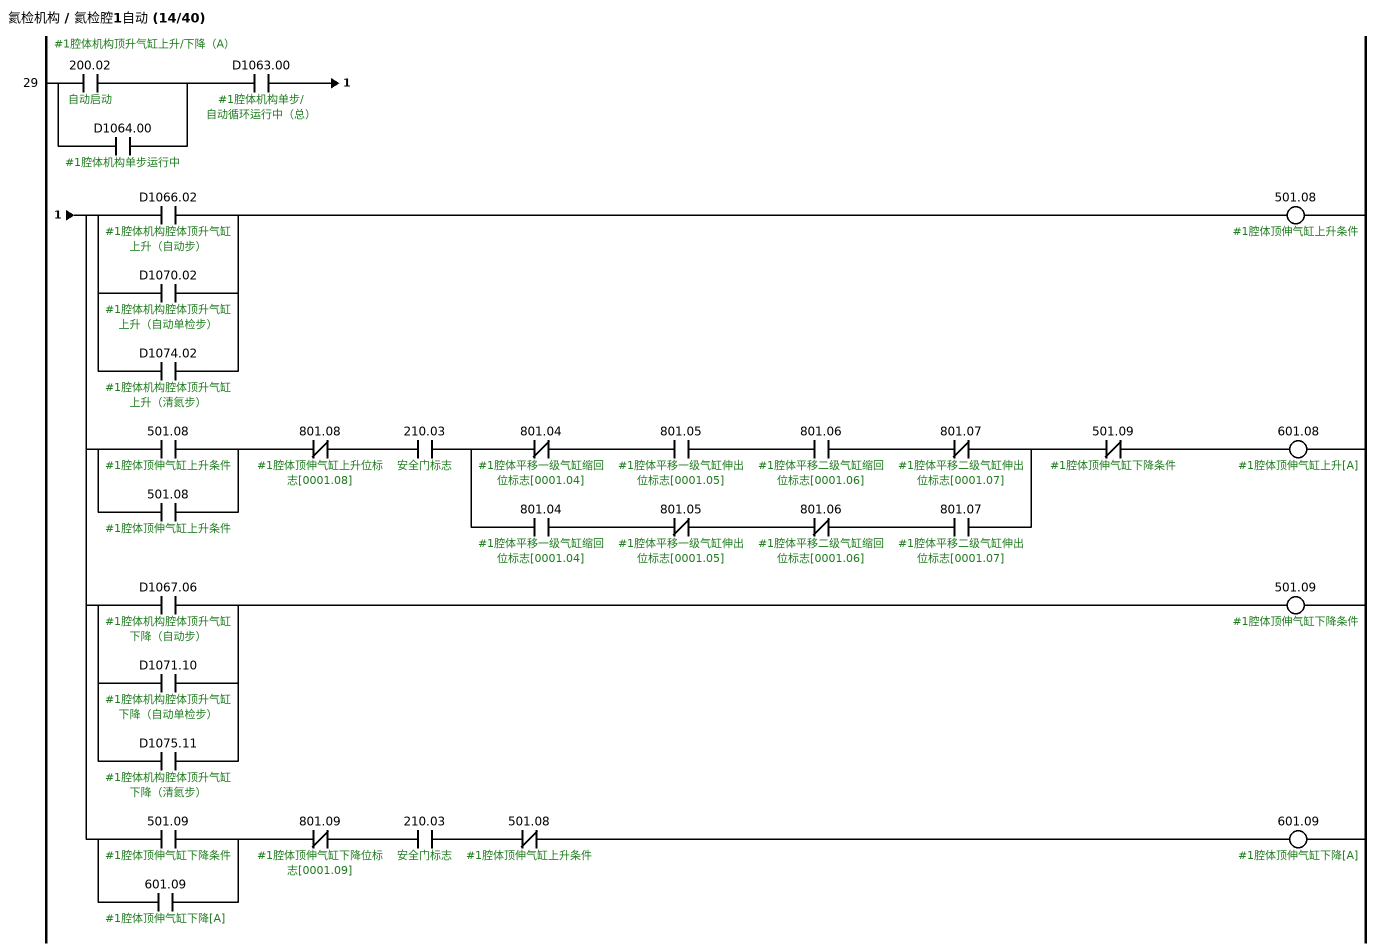
; [picture p216: 氦检机构 / 氦检腔1自动, rungs 29-29]
; rung 29: #1腔体机构顶升气缸上升/下降（A）
LD 200.02  ; 自动启动
OR D1064.00  ; #1腔体机构单步运行中
AND D1063.00  ; #1腔体机构单步/自动循环运行中（总）
OUT TR0
LD D1066.02  ; #1腔体机构腔体顶升气缸上升（自动步）
OR D1070.02  ; #1腔体机构腔体顶升气缸上升（自动单检步）
OR D1074.02  ; #1腔体机构腔体顶升气缸上升（清氦步）
ANDLD
OUT 501.08  ; #1腔体顶伸气缸上升条件
LD TR0
LD 501.08  ; #1腔体顶伸气缸上升条件
OR 501.08  ; #1腔体顶伸气缸上升条件
ANDLD
ANDNOT 801.08  ; #1腔体顶伸气缸上升位标志[0001.08]
AND 210.03  ; 安全门标志
LDNOT 801.04  ; #1腔体平移一级气缸缩回位标志[0001.04]
AND 801.05  ; #1腔体平移一级气缸伸出位标志[0001.05]
AND 801.06  ; #1腔体平移二级气缸缩回位标志[0001.06]
ANDNOT 801.07  ; #1腔体平移二级气缸伸出位标志[0001.07]
LD 801.04  ; #1腔体平移一级气缸缩回位标志[0001.04]
ANDNOT 801.05  ; #1腔体平移一级气缸伸出位标志[0001.05]
ANDNOT 801.06  ; #1腔体平移二级气缸缩回位标志[0001.06]
AND 801.07  ; #1腔体平移二级气缸伸出位标志[0001.07]
ORLD
ANDLD
ANDNOT 501.09  ; #1腔体顶伸气缸下降条件
OUT 601.08  ; #1腔体顶伸气缸上升[A]
LD TR0
LD D1067.06  ; #1腔体机构腔体顶升气缸下降（自动步）
OR D1071.10  ; #1腔体机构腔体顶升气缸下降（自动单检步）
OR D1075.11  ; #1腔体机构腔体顶升气缸下降（清氦步）
ANDLD
OUT 501.09  ; #1腔体顶伸气缸下降条件
LD TR0
LD 501.09  ; #1腔体顶伸气缸下降条件
OR 601.09  ; #1腔体顶伸气缸下降[A]
ANDLD
ANDNOT 801.09  ; #1腔体顶伸气缸下降位标志[0001.09]
AND 210.03  ; 安全门标志
ANDNOT 501.08  ; #1腔体顶伸气缸上升条件
OUT 601.09  ; #1腔体顶伸气缸下降[A]

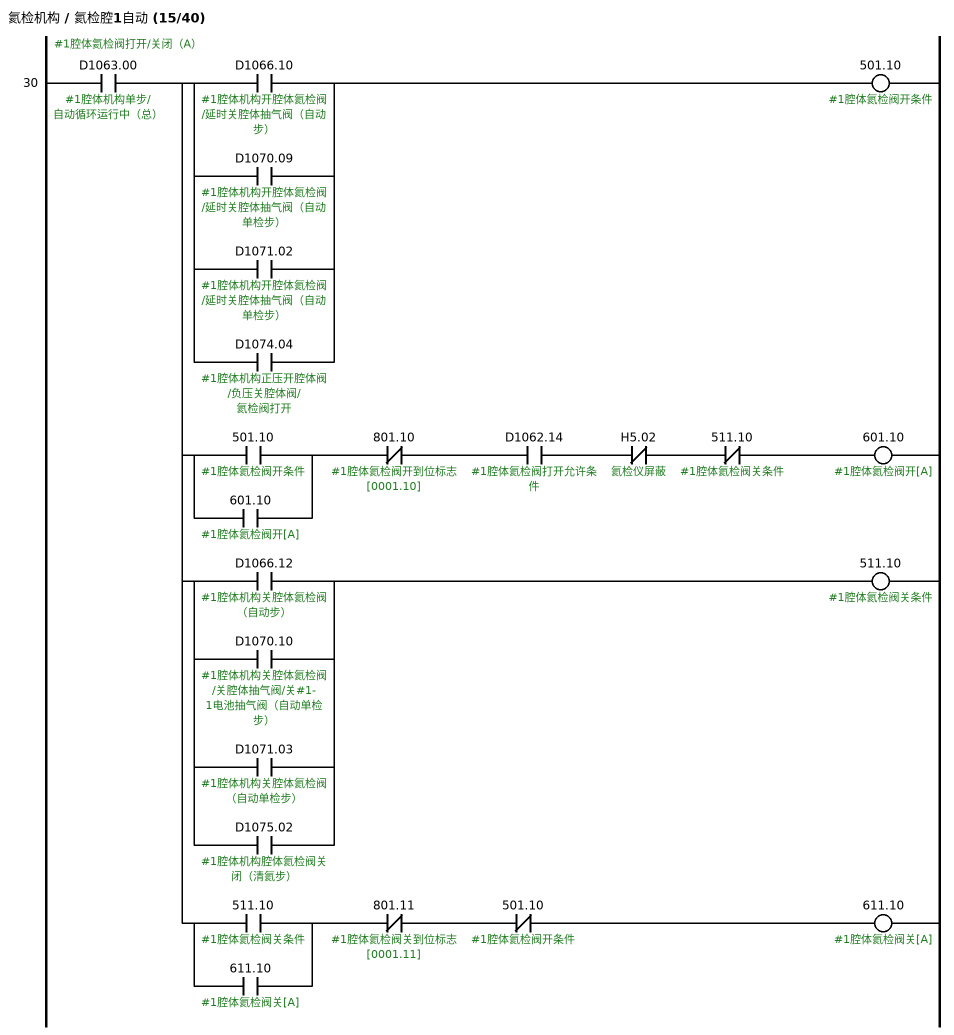
; rung 30: #1腔体氦检阀打开/关闭（A）
LD D1063.00  ; #1腔体机构单步/自动循环运行中（总）
OUT TR0
LD D1066.10  ; #1腔体机构开腔体氦检阀/延时关腔体抽气阀（自动步）
OR D1070.09  ; #1腔体机构开腔体氦检阀/延时关腔体抽气阀（自动单检步）
OR D1071.02  ; #1腔体机构开腔体氦检阀/延时关腔体抽气阀（自动单检步）
OR D1074.04  ; #1腔体机构正压开腔体阀/负压关腔体阀/氦检阀打开
ANDLD
OUT 501.10  ; #1腔体氦检阀开条件
LD TR0
LD 501.10  ; #1腔体氦检阀开条件
OR 601.10  ; #1腔体氦检阀开[A]
ANDLD
ANDNOT 801.10  ; #1腔体氦检阀开到位标志[0001.10]
AND D1062.14  ; #1腔体氦检阀打开允许条件
ANDNOT H5.02  ; 氦检仪屏蔽
ANDNOT 511.10  ; #1腔体氦检阀关条件
OUT 601.10  ; #1腔体氦检阀开[A]
LD TR0
LD D1066.12  ; #1腔体机构关腔体氦检阀（自动步）
OR D1070.10  ; #1腔体机构关腔体氦检阀/关腔体抽气阀/关#1-1电池抽气阀（自动单检步）
OR D1071.03  ; #1腔体机构关腔体氦检阀（自动单检步）
OR D1075.02  ; #1腔体机构腔体氦检阀关闭（清氦步）
ANDLD
OUT 511.10  ; #1腔体氦检阀关条件
LD TR0
LD 511.10  ; #1腔体氦检阀关条件
OR 611.10  ; #1腔体氦检阀关[A]
ANDLD
ANDNOT 801.11  ; #1腔体氦检阀关到位标志[0001.11]
ANDNOT 501.10  ; #1腔体氦检阀开条件
OUT 611.10  ; #1腔体氦检阀关[A]

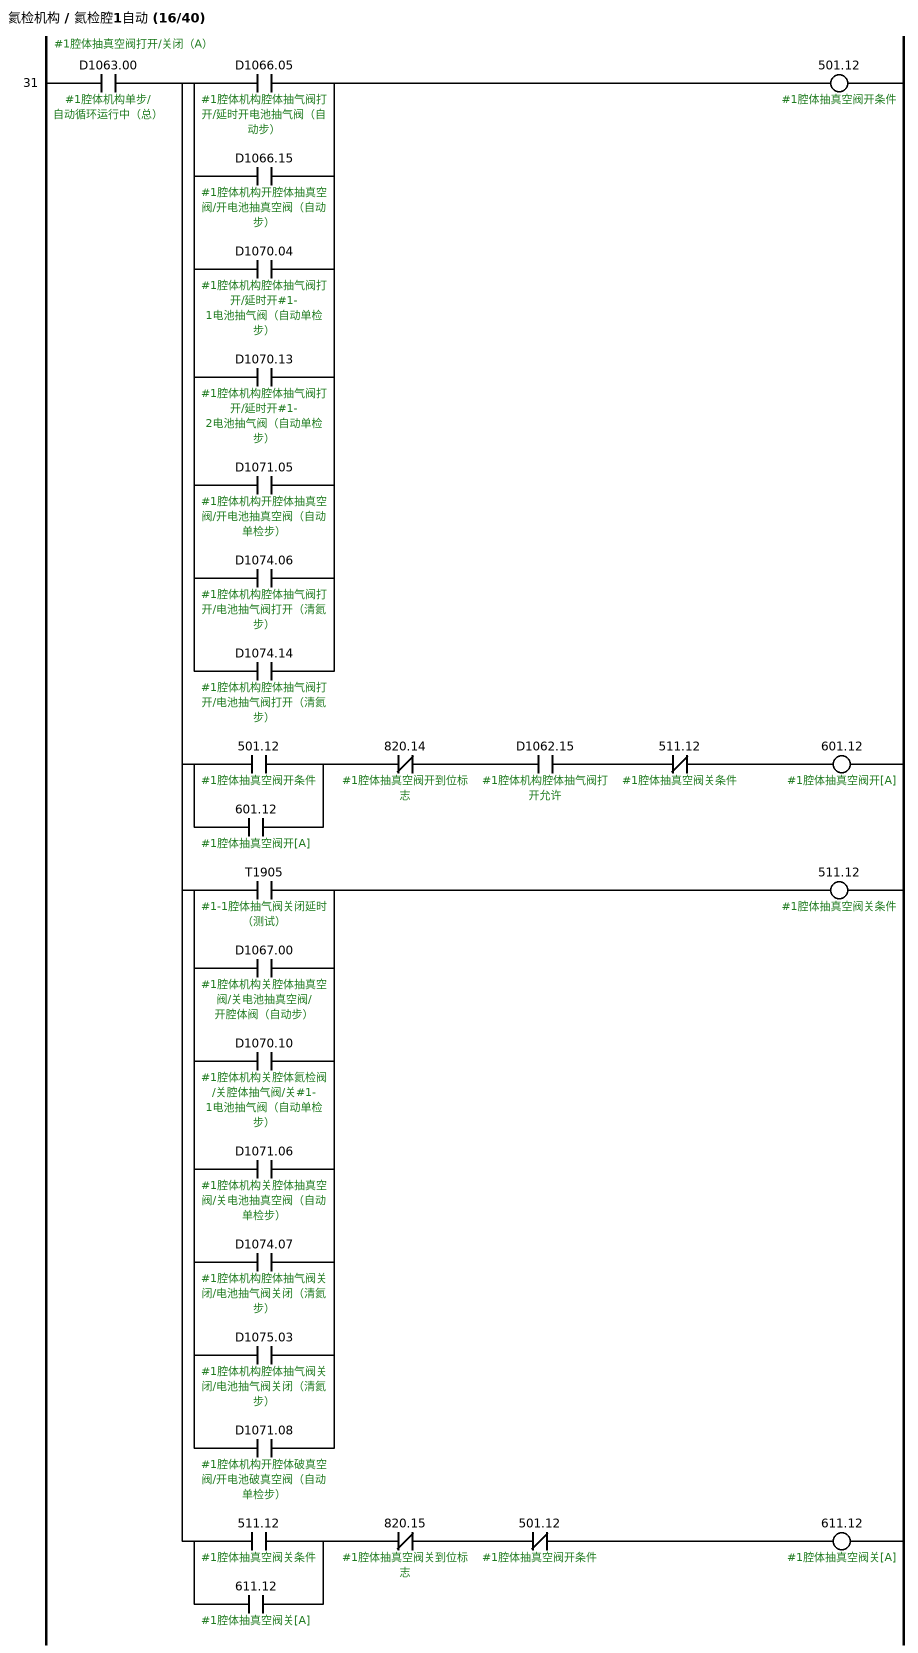
; rung 31: #1腔体抽真空阀打开/关闭（A）
LD D1063.00  ; #1腔体机构单步/自动循环运行中（总）
OUT TR0
LD D1066.05  ; #1腔体机构腔体抽气阀打开/延时开电池抽气阀（自动步）
OR D1066.15  ; #1腔体机构开腔体抽真空阀/开电池抽真空阀（自动步）
OR D1070.04  ; #1腔体机构腔体抽气阀打开/延时开#1-1电池抽气阀（自动单检步）
OR D1070.13  ; #1腔体机构腔体抽气阀打开/延时开#1-2电池抽气阀（自动单检步）
OR D1071.05  ; #1腔体机构开腔体抽真空阀/开电池抽真空阀（自动单检步）
OR D1074.06  ; #1腔体机构腔体抽气阀打开/电池抽气阀打开（清氦步）
OR D1074.14  ; #1腔体机构腔体抽气阀打开/电池抽气阀打开（清氦步）
ANDLD
OUT 501.12  ; #1腔体抽真空阀开条件
LD TR0
LD 501.12  ; #1腔体抽真空阀开条件
OR 601.12  ; #1腔体抽真空阀开[A]
ANDLD
ANDNOT 820.14  ; #1腔体抽真空阀开到位标志
AND D1062.15  ; #1腔体机构腔体抽气阀打开允许
ANDNOT 511.12  ; #1腔体抽真空阀关条件
OUT 601.12  ; #1腔体抽真空阀开[A]
LD TR0
LD T1905  ; #1-1腔体抽气阀关闭延时（测试）
OR D1067.00  ; #1腔体机构关腔体抽真空阀/关电池抽真空阀/开腔体阀（自动步）
OR D1070.10  ; #1腔体机构关腔体氦检阀/关腔体抽气阀/关#1-1电池抽气阀（自动单检步）
OR D1071.06  ; #1腔体机构关腔体抽真空阀/关电池抽真空阀（自动单检步）
OR D1074.07  ; #1腔体机构腔体抽气阀关闭/电池抽气阀关闭（清氦步）
OR D1075.03  ; #1腔体机构腔体抽气阀关闭/电池抽气阀关闭（清氦步）
OR D1071.08  ; #1腔体机构开腔体破真空阀/开电池破真空阀（自动单检步）
ANDLD
OUT 511.12  ; #1腔体抽真空阀关条件
LD TR0
LD 511.12  ; #1腔体抽真空阀关条件
OR 611.12  ; #1腔体抽真空阀关[A]
ANDLD
ANDNOT 820.15  ; #1腔体抽真空阀关到位标志
ANDNOT 501.12  ; #1腔体抽真空阀开条件
OUT 611.12  ; #1腔体抽真空阀关[A]

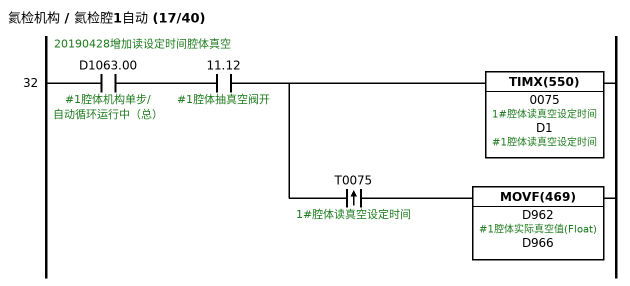
; rung 32: 20190428增加读设定时间腔体真空
LD D1063.00  ; #1腔体机构单步/自动循环运行中（总）
AND 11.12  ; #1腔体抽真空阀开
TIMX(550) 0075 D1  ; #1腔体读真空设定时间, 1#腔体读真空设定时间
@AND T0075  ; 1#腔体读真空设定时间
MOVF(469) D962 D966  ; #1腔体实际真空值(Float)

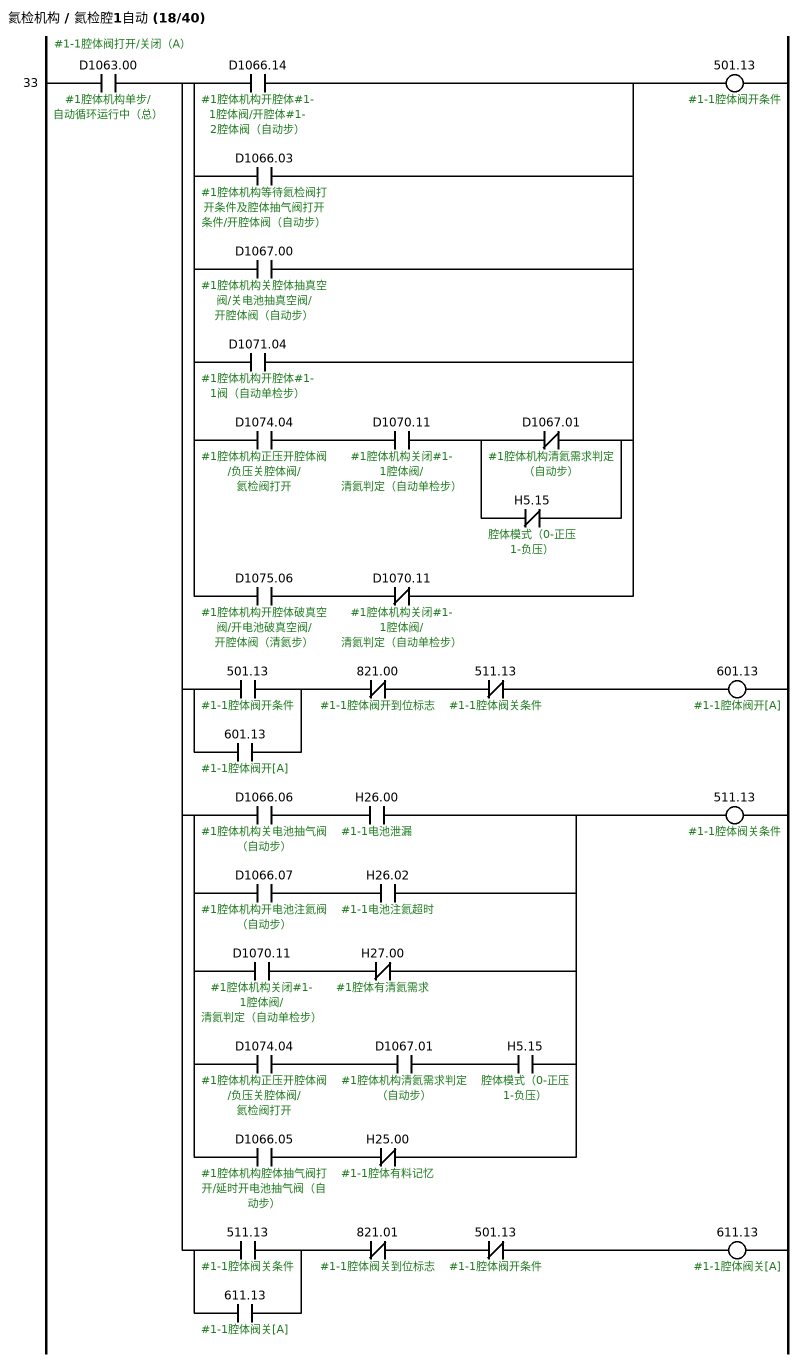
; rung 33: #1-1腔体阀打开/关闭（A）
LD D1063.00  ; #1腔体机构单步/自动循环运行中（总）
OUT TR0
LD D1066.14  ; #1腔体机构开腔体#1-1腔体阀/开腔体#1-2腔体阀（自动步）
OR D1066.03  ; #1腔体机构等待氦检阀打开条件及腔体抽气阀打开条件/开腔体阀（自动步）
OR D1067.00  ; #1腔体机构关腔体抽真空阀/关电池抽真空阀/开腔体阀（自动步）
OR D1071.04  ; #1腔体机构开腔体#1-1阀（自动单检步）
LD D1074.04  ; #1腔体机构正压开腔体阀/负压关腔体阀/氦检阀打开
AND D1070.11  ; #1腔体机构关闭#1-1腔体阀/清氦判定（自动单检步）
LDNOT D1067.01  ; #1腔体机构清氦需求判定（自动步）
ORNOT H5.15  ; 腔体模式（0-正压 1-负压）
ANDLD
ORLD
LD D1075.06  ; #1腔体机构开腔体破真空阀/开电池破真空阀/开腔体阀（清氦步）
ANDNOT D1070.11  ; #1腔体机构关闭#1-1腔体阀/清氦判定（自动单检步）
ORLD
ANDLD
OUT 501.13  ; #1-1腔体阀开条件
LD TR0
LD 501.13  ; #1-1腔体阀开条件
OR 601.13  ; #1-1腔体阀开[A]
ANDLD
ANDNOT 821.00  ; #1-1腔体阀开到位标志
ANDNOT 511.13  ; #1-1腔体阀关条件
OUT 601.13  ; #1-1腔体阀开[A]
LD TR0
LD D1066.06  ; #1腔体机构关电池抽气阀（自动步）
AND H26.00  ; #1-1电池泄漏
LD D1066.07  ; #1腔体机构开电池注氦阀（自动步）
AND H26.02  ; #1-1电池注氦超时
ORLD
LD D1070.11  ; #1腔体机构关闭#1-1腔体阀/清氦判定（自动单检步）
ANDNOT H27.00  ; #1腔体有清氦需求
ORLD
LD D1074.04  ; #1腔体机构正压开腔体阀/负压关腔体阀/氦检阀打开
AND D1067.01  ; #1腔体机构清氦需求判定（自动步）
AND H5.15  ; 腔体模式（0-正压 1-负压）
ORLD
LD D1066.05  ; #1腔体机构腔体抽气阀打开/延时开电池抽气阀（自动步）  // #1-1无料时不测试
ANDNOT H25.00  ; #1-1腔体有料记忆
ORLD
ANDLD
OUT 511.13  ; #1-1腔体阀关条件
LD TR0
LD 511.13  ; #1-1腔体阀关条件
OR 611.13  ; #1-1腔体阀关[A]
ANDLD
ANDNOT 821.01  ; #1-1腔体阀关到位标志
ANDNOT 501.13  ; #1-1腔体阀开条件
OUT 611.13  ; #1-1腔体阀关[A]

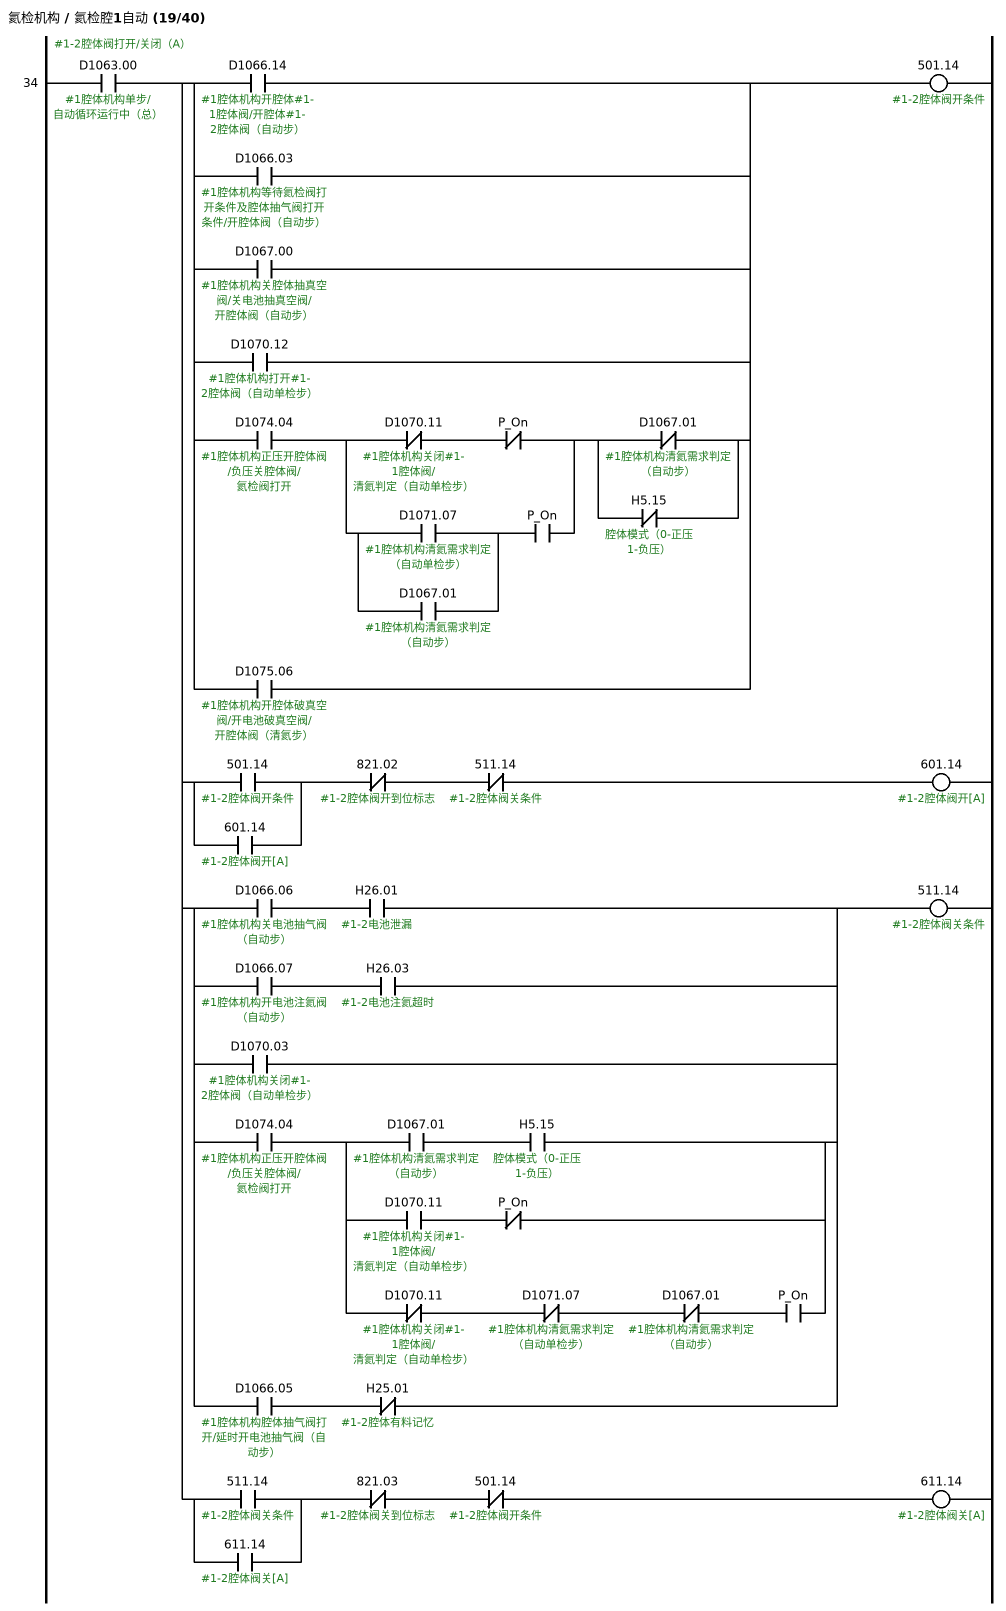
; rung 34: #1-2腔体阀打开/关闭（A）
LD D1063.00  ; #1腔体机构单步/自动循环运行中（总）
OUT TR0
LD D1066.14  ; #1腔体机构开腔体#1-1腔体阀/开腔体#1-2腔体阀（自动步）
OR D1066.03  ; #1腔体机构等待氦检阀打开条件及腔体抽气阀打开条件/开腔体阀（自动步）
OR D1067.00  ; #1腔体机构关腔体抽真空阀/关电池抽真空阀/开腔体阀（自动步）
OR D1070.12  ; #1腔体机构打开#1-2腔体阀（自动单检步）
LD D1074.04  ; #1腔体机构正压开腔体阀/负压关腔体阀/氦检阀打开
LDNOT D1070.11  ; #1腔体机构关闭#1-1腔体阀/清氦判定（自动单检步）
ANDNOT P_On
LD D1071.07  ; #1腔体机构清氦需求判定（自动单检步）
OR D1067.01  ; #1腔体机构清氦需求判定（自动步）
AND P_On
ORLD
ANDLD
LDNOT D1067.01  ; #1腔体机构清氦需求判定（自动步）
ORNOT H5.15  ; 腔体模式（0-正压 1-负压）
ANDLD
ORLD
OR D1075.06  ; #1腔体机构开腔体破真空阀/开电池破真空阀/开腔体阀（清氦步）
ANDLD
OUT 501.14  ; #1-2腔体阀开条件
LD TR0
LD 501.14  ; #1-2腔体阀开条件
OR 601.14  ; #1-2腔体阀开[A]
ANDLD
ANDNOT 821.02  ; #1-2腔体阀开到位标志
ANDNOT 511.14  ; #1-2腔体阀关条件
OUT 601.14  ; #1-2腔体阀开[A]
LD TR0
LD D1066.06  ; #1腔体机构关电池抽气阀（自动步）
AND H26.01  ; #1-2电池泄漏
LD D1066.07  ; #1腔体机构开电池注氦阀（自动步）
AND H26.03  ; #1-2电池注氦超时
ORLD
OR D1070.03  ; #1腔体机构关闭#1-2腔体阀（自动单检步）
LD D1074.04  ; #1腔体机构正压开腔体阀/负压关腔体阀/氦检阀打开
LD D1067.01  ; #1腔体机构清氦需求判定（自动步）
AND H5.15  ; 腔体模式（0-正压 1-负压）
LD D1070.11  ; #1腔体机构关闭#1-1腔体阀/清氦判定（自动单检步）
ANDNOT P_On
ORLD
LDNOT D1070.11  ; #1腔体机构关闭#1-1腔体阀/清氦判定（自动单检步）
ANDNOT D1071.07  ; #1腔体机构清氦需求判定（自动单检步）
ANDNOT D1067.01  ; #1腔体机构清氦需求判定（自动步）
AND P_On
ORLD
ANDLD
ORLD
LD D1066.05  ; #1腔体机构腔体抽气阀打开/延时开电池抽气阀（自动步）  // #1-2无料时不测试
ANDNOT H25.01  ; #1-2腔体有料记忆
ORLD
ANDLD
OUT 511.14  ; #1-2腔体阀关条件
LD TR0
LD 511.14  ; #1-2腔体阀关条件
OR 611.14  ; #1-2腔体阀关[A]
ANDLD
ANDNOT 821.03  ; #1-2腔体阀关到位标志
ANDNOT 501.14  ; #1-2腔体阀开条件
OUT 611.14  ; #1-2腔体阀关[A]

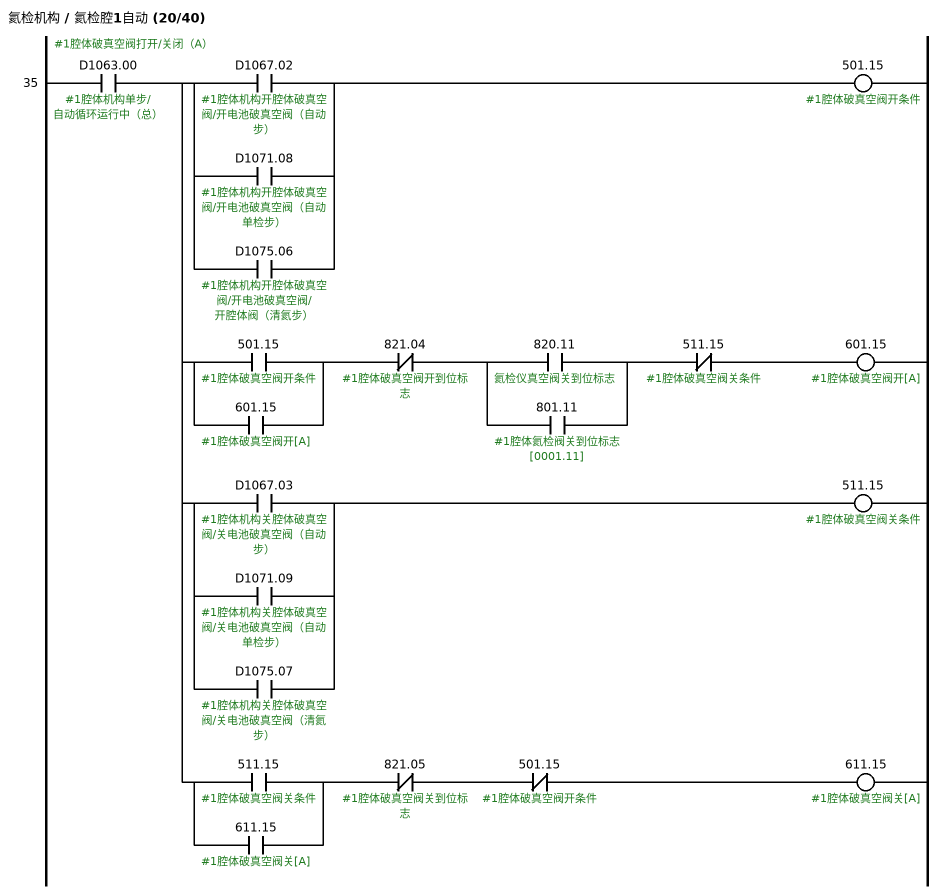
; rung 35: #1腔体破真空阀打开/关闭（A）
LD D1063.00  ; #1腔体机构单步/自动循环运行中（总）
OUT TR0
LD D1067.02  ; #1腔体机构开腔体破真空阀/开电池破真空阀（自动步）
OR D1071.08  ; #1腔体机构开腔体破真空阀/开电池破真空阀（自动单检步）
OR D1075.06  ; #1腔体机构开腔体破真空阀/开电池破真空阀/开腔体阀（清氦步）
ANDLD
OUT 501.15  ; #1腔体破真空阀开条件
LD TR0
LD 501.15  ; #1腔体破真空阀开条件
OR 601.15  ; #1腔体破真空阀开[A]
ANDLD
ANDNOT 821.04  ; #1腔体破真空阀开到位标志
LD 820.11  ; 氦检仪真空阀关到位标志
OR 801.11  ; #1腔体氦检阀关到位标志[0001.11]
ANDLD
ANDNOT 511.15  ; #1腔体破真空阀关条件
OUT 601.15  ; #1腔体破真空阀开[A]
LD TR0
LD D1067.03  ; #1腔体机构关腔体破真空阀/关电池破真空阀（自动步）
OR D1071.09  ; #1腔体机构关腔体破真空阀/关电池破真空阀（自动单检步）
OR D1075.07  ; #1腔体机构关腔体破真空阀/关电池破真空阀（清氦步）
ANDLD
OUT 511.15  ; #1腔体破真空阀关条件
LD TR0
LD 511.15  ; #1腔体破真空阀关条件
OR 611.15  ; #1腔体破真空阀关[A]
ANDLD
ANDNOT 821.05  ; #1腔体破真空阀关到位标志
ANDNOT 501.15  ; #1腔体破真空阀开条件
OUT 611.15  ; #1腔体破真空阀关[A]

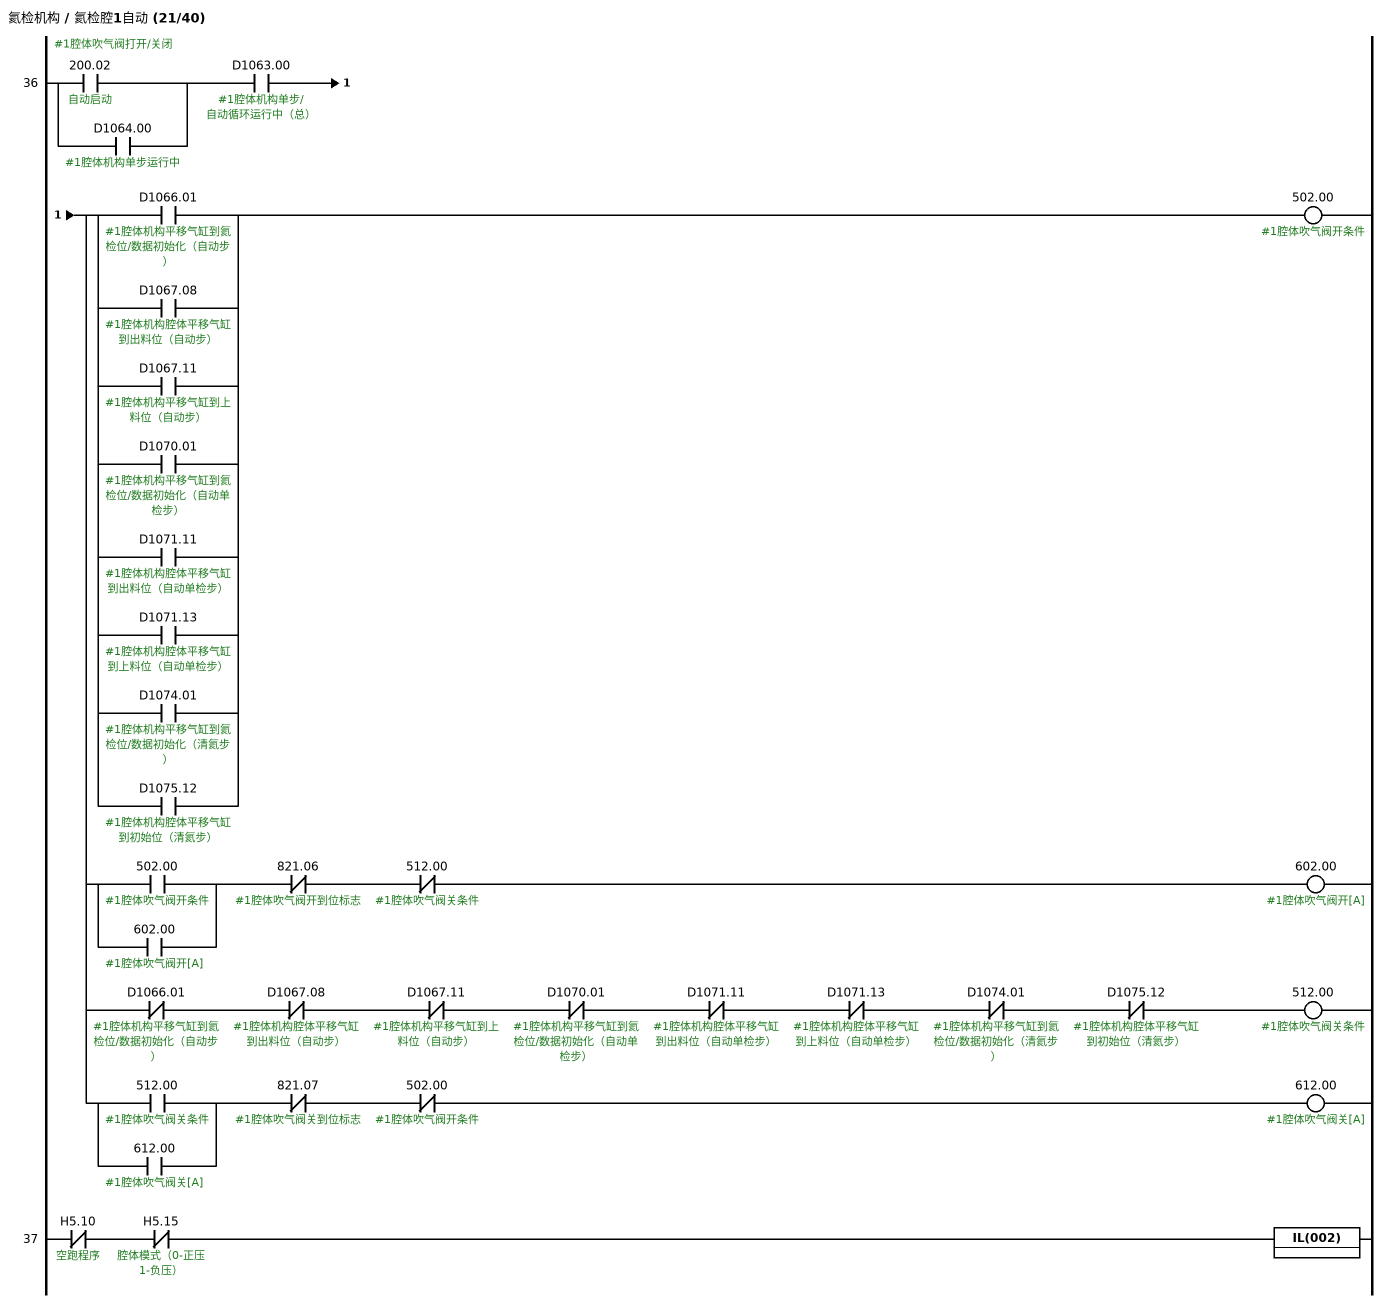
; rung 36: #1腔体吹气阀打开/关闭
LD 200.02  ; 自动启动
OR D1064.00  ; #1腔体机构单步运行中
AND D1063.00  ; #1腔体机构单步/自动循环运行中（总）
OUT TR0
LD D1066.01  ; #1腔体机构平移气缸到氦检位/数据初始化（自动步）
OR D1067.08  ; #1腔体机构腔体平移气缸到出料位（自动步）
OR D1067.11  ; #1腔体机构平移气缸到上料位（自动步）
OR D1070.01  ; #1腔体机构平移气缸到氦检位/数据初始化（自动单检步）
OR D1071.11  ; #1腔体机构腔体平移气缸到出料位（自动单检步）
OR D1071.13  ; #1腔体机构腔体平移气缸到上料位（自动单检步）
OR D1074.01  ; #1腔体机构平移气缸到氦检位/数据初始化（清氦步）
OR D1075.12  ; #1腔体机构腔体平移气缸到初始位（清氦步）
ANDLD
OUT 502.00  ; #1腔体吹气阀开条件
LD TR0
LD 502.00  ; #1腔体吹气阀开条件
OR 602.00  ; #1腔体吹气阀开[A]
ANDLD
ANDNOT 821.06  ; #1腔体吹气阀开到位标志
ANDNOT 512.00  ; #1腔体吹气阀关条件
OUT 602.00  ; #1腔体吹气阀开[A]
LD TR0
ANDNOT D1066.01  ; #1腔体机构平移气缸到氦检位/数据初始化（自动步）
ANDNOT D1067.08  ; #1腔体机构腔体平移气缸到出料位（自动步）
ANDNOT D1067.11  ; #1腔体机构平移气缸到上料位（自动步）
ANDNOT D1070.01  ; #1腔体机构平移气缸到氦检位/数据初始化（自动单检步）
ANDNOT D1071.11  ; #1腔体机构腔体平移气缸到出料位（自动单检步）
ANDNOT D1071.13  ; #1腔体机构腔体平移气缸到上料位（自动单检步）
ANDNOT D1074.01  ; #1腔体机构平移气缸到氦检位/数据初始化（清氦步）
ANDNOT D1075.12  ; #1腔体机构腔体平移气缸到初始位（清氦步）
OUT 512.00  ; #1腔体吹气阀关条件
LD TR0
LD 512.00  ; #1腔体吹气阀关条件
OR 612.00  ; #1腔体吹气阀关[A]
ANDLD
ANDNOT 821.07  ; #1腔体吹气阀关到位标志
ANDNOT 502.00  ; #1腔体吹气阀开条件
OUT 612.00  ; #1腔体吹气阀关[A]
; rung 37
LDNOT H5.10  ; 空跑程序
ANDNOT H5.15  ; 腔体模式（0-正压 1-负压）
IL(002)

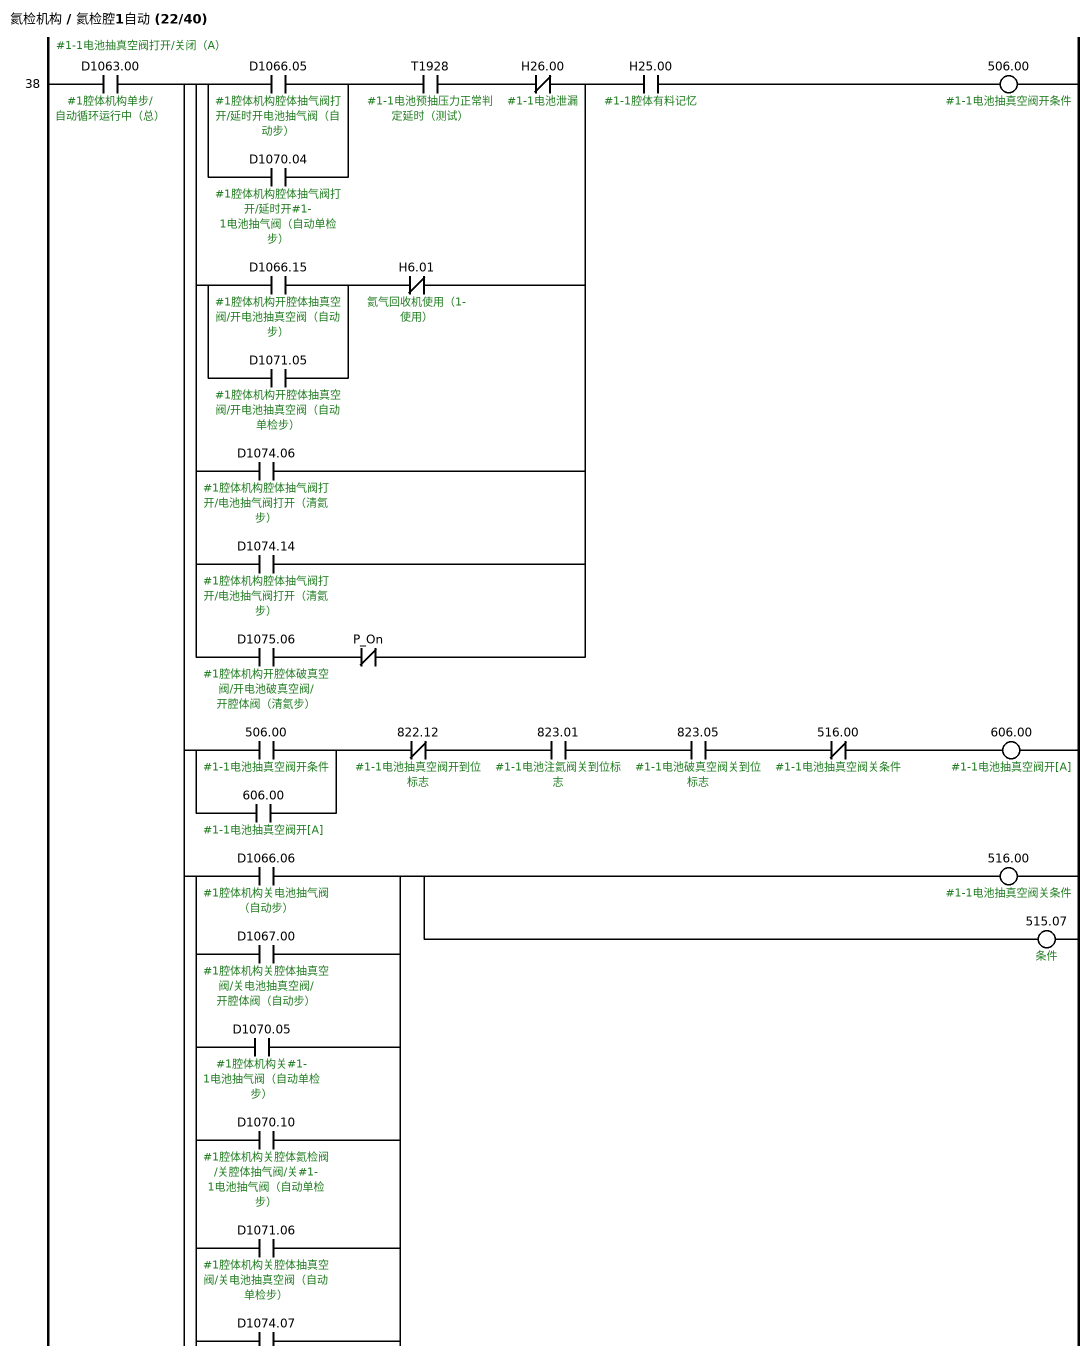

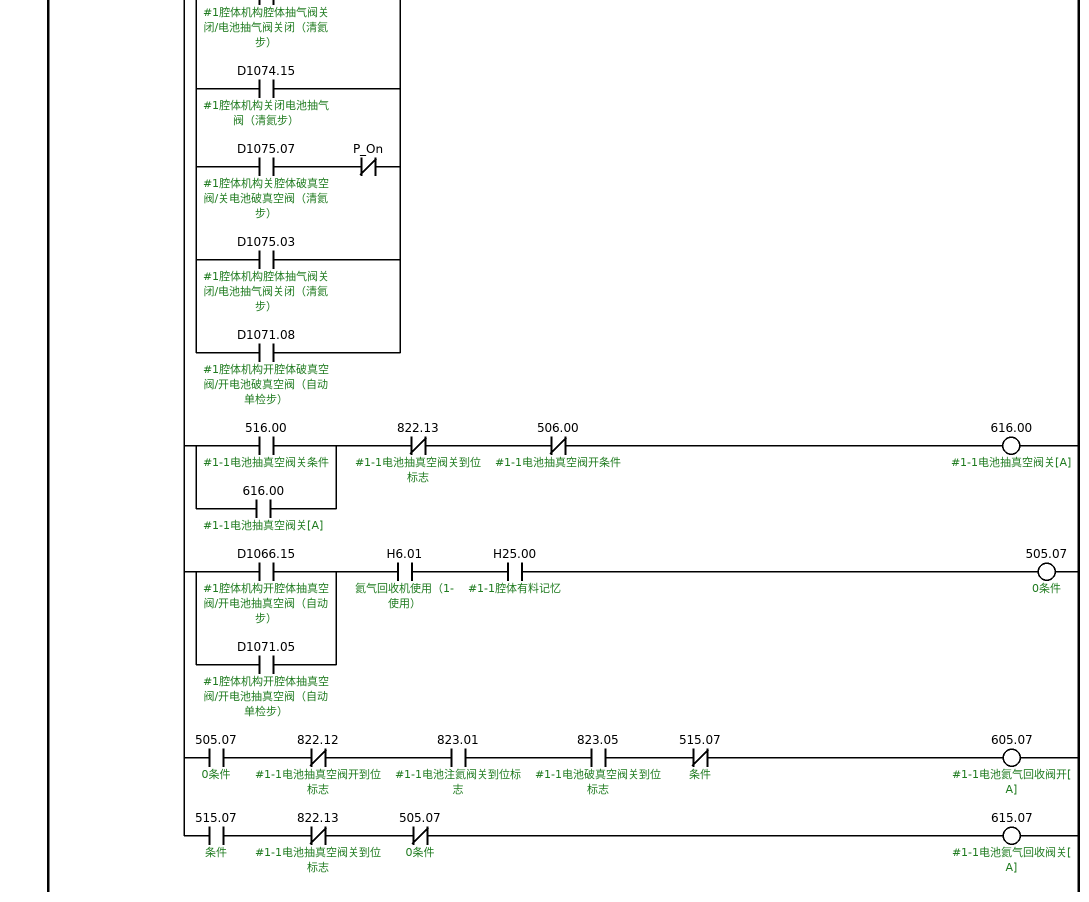
; rung 38: #1-1电池抽真空阀打开/关闭（A）
LD D1063.00  ; #1腔体机构单步/自动循环运行中（总）
OUT TR0
LD D1066.05  ; #1腔体机构腔体抽气阀打开/延时开电池抽气阀（自动步）
OR D1070.04  ; #1腔体机构腔体抽气阀打开/延时开#1-1电池抽气阀（自动单检步）
AND T1928  ; #1-1电池预抽压力正常判定延时（测试）
ANDNOT H26.00  ; #1-1电池泄漏
LD D1066.15  ; #1腔体机构开腔体抽真空阀/开电池抽真空阀（自动步）
OR D1071.05  ; #1腔体机构开腔体抽真空阀/开电池抽真空阀（自动单检步）
ANDNOT H6.01  ; 氦气回收机使用（1-使用）
ORLD
OR D1074.06  ; #1腔体机构腔体抽气阀打开/电池抽气阀打开（清氦步）
OR D1074.14  ; #1腔体机构腔体抽气阀打开/电池抽气阀打开（清氦步）
LD D1075.06  ; #1腔体机构开腔体破真空阀/开电池破真空阀/开腔体阀（清氦步）
ANDNOT P_On
ORLD
ANDLD
AND H25.00  ; #1-1腔体有料记忆
OUT 506.00  ; #1-1电池抽真空阀开条件
LD TR0
LD 506.00  ; #1-1电池抽真空阀开条件
OR 606.00  ; #1-1电池抽真空阀开[A]
ANDLD
ANDNOT 822.12  ; #1-1电池抽真空阀开到位标志
AND 823.01  ; #1-1电池注氦阀关到位标志
AND 823.05  ; #1-1电池破真空阀关到位标志
ANDNOT 516.00  ; #1-1电池抽真空阀关条件
OUT 606.00  ; #1-1电池抽真空阀开[A]
LD TR0
LD D1066.06  ; #1腔体机构关电池抽气阀（自动步）
OR D1067.00  ; #1腔体机构关腔体抽真空阀/关电池抽真空阀/开腔体阀（自动步）
OR D1070.05  ; #1腔体机构关#1-1电池抽气阀（自动单检步）
OR D1070.10  ; #1腔体机构关腔体氦检阀/关腔体抽气阀/关#1-1电池抽气阀（自动单检步）
OR D1071.06  ; #1腔体机构关腔体抽真空阀/关电池抽真空阀（自动单检步）
OR D1074.07  ; #1腔体机构腔体抽气阀关闭/电池抽气阀关闭（清氦步）
OR D1074.15  ; #1腔体机构关闭电池抽气阀（清氦步）
LD D1075.07  ; #1腔体机构关腔体破真空阀/关电池破真空阀（清氦步）
ANDNOT P_On
ORLD
OR D1075.03  ; #1腔体机构腔体抽气阀关闭/电池抽气阀关闭（清氦步）
OR D1071.08  ; #1腔体机构开腔体破真空阀/开电池破真空阀（自动单检步）
ANDLD
OUT 516.00  ; #1-1电池抽真空阀关条件
OUT 515.07  ; 条件
LD TR0
LD 516.00  ; #1-1电池抽真空阀关条件
OR 616.00  ; #1-1电池抽真空阀关[A]
ANDLD
ANDNOT 822.13  ; #1-1电池抽真空阀关到位标志
ANDNOT 506.00  ; #1-1电池抽真空阀开条件
OUT 616.00  ; #1-1电池抽真空阀关[A]
LD TR0
LD D1066.15  ; #1腔体机构开腔体抽真空阀/开电池抽真空阀（自动步）
OR D1071.05  ; #1腔体机构开腔体抽真空阀/开电池抽真空阀（自动单检步）
ANDLD
AND H6.01  ; 氦气回收机使用（1-使用）
AND H25.00  ; #1-1腔体有料记忆
OUT 505.07  ; 0条件
LD TR0
AND 505.07  ; 0条件
ANDNOT 822.12  ; #1-1电池抽真空阀开到位标志
AND 823.01  ; #1-1电池注氦阀关到位标志
AND 823.05  ; #1-1电池破真空阀关到位标志
ANDNOT 515.07  ; 条件
OUT 605.07  ; #1-1电池氦气回收阀开[A]
LD TR0
AND 515.07  ; 条件
ANDNOT 822.13  ; #1-1电池抽真空阀关到位标志
ANDNOT 505.07  ; 0条件
OUT 615.07  ; #1-1电池氦气回收阀关[A]

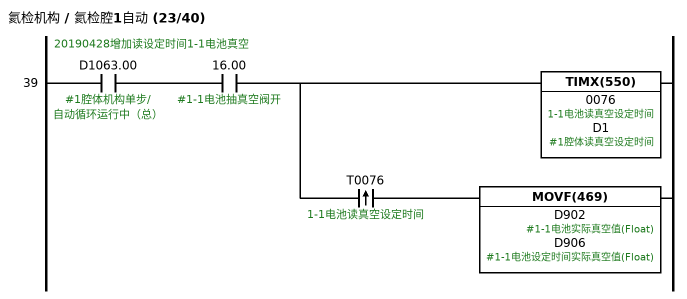
; rung 39: 20190428增加读设定时间1-1电池真空
LD D1063.00  ; #1腔体机构单步/自动循环运行中（总）
AND 16.00  ; #1-1电池抽真空阀开
TIMX(550) 0076 D1  ; #1腔体读真空设定时间, 1-1电池读真空设定时间
@AND T0076  ; 1-1电池读真空设定时间
MOVF(469) D902 D906  ; #1-1电池实际真空值(Float), #1-1电池设定时间实际真空值(Float)

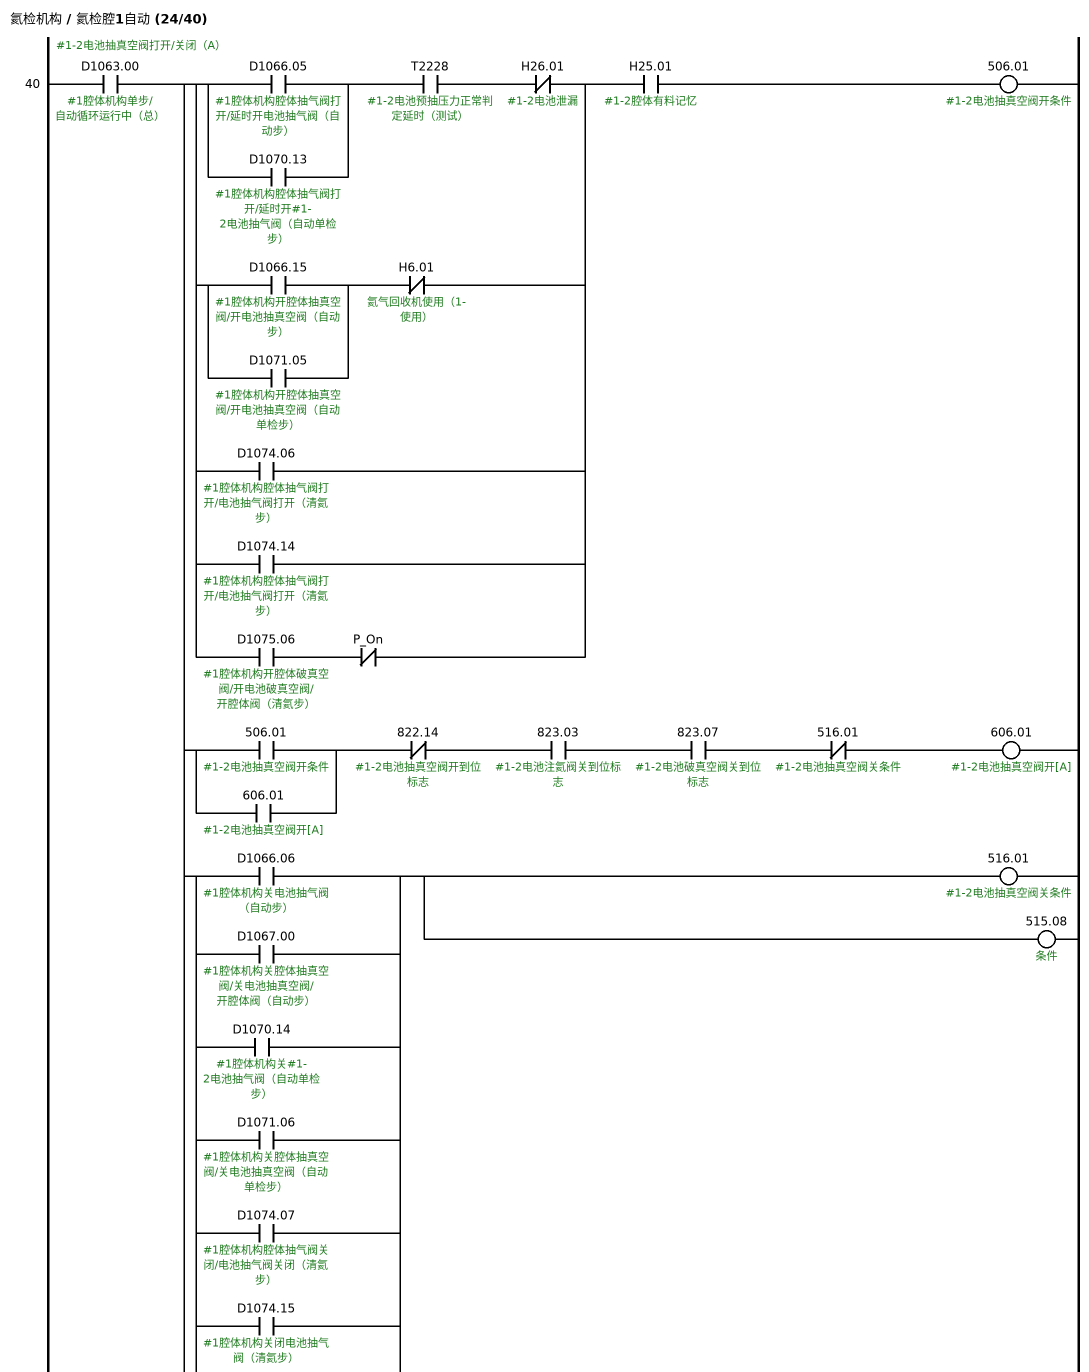

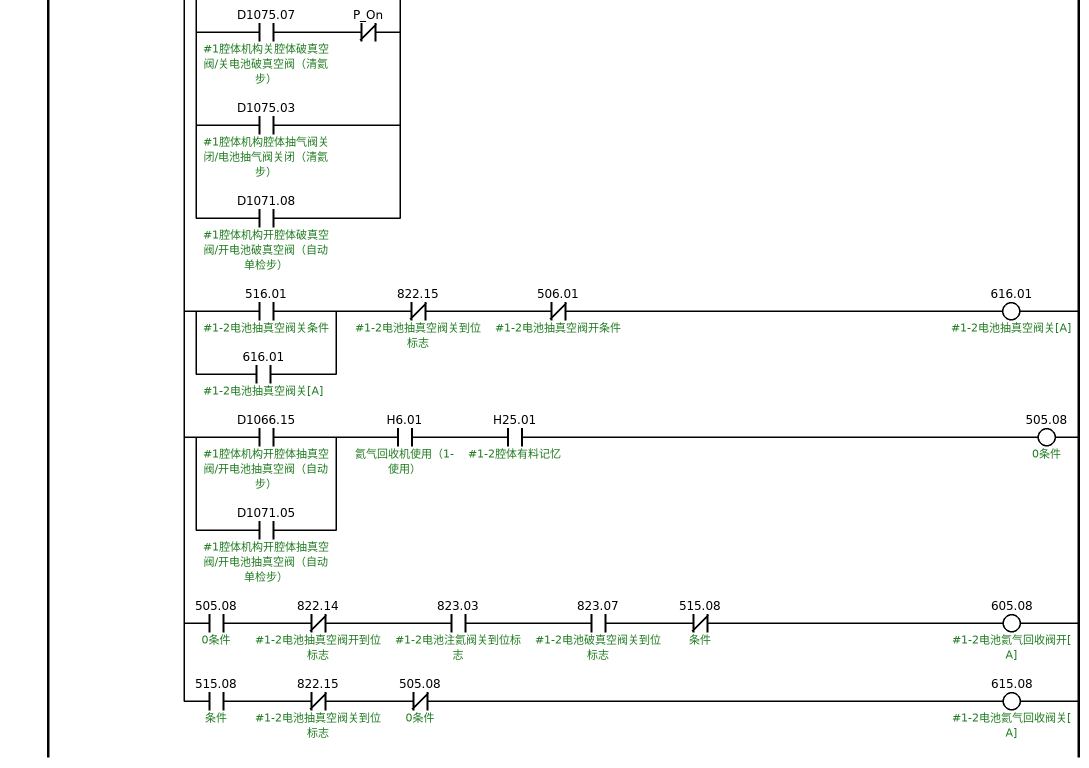
; rung 40: #1-2电池抽真空阀打开/关闭（A）
LD D1063.00  ; #1腔体机构单步/自动循环运行中（总）
OUT TR0
LD D1066.05  ; #1腔体机构腔体抽气阀打开/延时开电池抽气阀（自动步）
OR D1070.13  ; #1腔体机构腔体抽气阀打开/延时开#1-2电池抽气阀（自动单检步）
AND T2228  ; #1-2电池预抽压力正常判定延时（测试）
ANDNOT H26.01  ; #1-2电池泄漏
LD D1066.15  ; #1腔体机构开腔体抽真空阀/开电池抽真空阀（自动步）
OR D1071.05  ; #1腔体机构开腔体抽真空阀/开电池抽真空阀（自动单检步）
ANDNOT H6.01  ; 氦气回收机使用（1-使用）
ORLD
OR D1074.06  ; #1腔体机构腔体抽气阀打开/电池抽气阀打开（清氦步）
OR D1074.14  ; #1腔体机构腔体抽气阀打开/电池抽气阀打开（清氦步）
LD D1075.06  ; #1腔体机构开腔体破真空阀/开电池破真空阀/开腔体阀（清氦步）
ANDNOT P_On
ORLD
ANDLD
AND H25.01  ; #1-2腔体有料记忆
OUT 506.01  ; #1-2电池抽真空阀开条件
LD TR0
LD 506.01  ; #1-2电池抽真空阀开条件
OR 606.01  ; #1-2电池抽真空阀开[A]
ANDLD
ANDNOT 822.14  ; #1-2电池抽真空阀开到位标志
AND 823.03  ; #1-2电池注氦阀关到位标志
AND 823.07  ; #1-2电池破真空阀关到位标志
ANDNOT 516.01  ; #1-2电池抽真空阀关条件
OUT 606.01  ; #1-2电池抽真空阀开[A]
LD TR0
LD D1066.06  ; #1腔体机构关电池抽气阀（自动步）
OR D1067.00  ; #1腔体机构关腔体抽真空阀/关电池抽真空阀/开腔体阀（自动步）
OR D1070.14  ; #1腔体机构关#1-2电池抽气阀（自动单检步）
OR D1071.06  ; #1腔体机构关腔体抽真空阀/关电池抽真空阀（自动单检步）
OR D1074.07  ; #1腔体机构腔体抽气阀关闭/电池抽气阀关闭（清氦步）
OR D1074.15  ; #1腔体机构关闭电池抽气阀（清氦步）
LD D1075.07  ; #1腔体机构关腔体破真空阀/关电池破真空阀（清氦步）
ANDNOT P_On
ORLD
OR D1075.03  ; #1腔体机构腔体抽气阀关闭/电池抽气阀关闭（清氦步）
OR D1071.08  ; #1腔体机构开腔体破真空阀/开电池破真空阀（自动单检步）
ANDLD
OUT 516.01  ; #1-2电池抽真空阀关条件
OUT 515.08  ; 条件
LD TR0
LD 516.01  ; #1-2电池抽真空阀关条件
OR 616.01  ; #1-2电池抽真空阀关[A]
ANDLD
ANDNOT 822.15  ; #1-2电池抽真空阀关到位标志
ANDNOT 506.01  ; #1-2电池抽真空阀开条件
OUT 616.01  ; #1-2电池抽真空阀关[A]
LD TR0
LD D1066.15  ; #1腔体机构开腔体抽真空阀/开电池抽真空阀（自动步）
OR D1071.05  ; #1腔体机构开腔体抽真空阀/开电池抽真空阀（自动单检步）
ANDLD
AND H6.01  ; 氦气回收机使用（1-使用）
AND H25.01  ; #1-2腔体有料记忆
OUT 505.08  ; 0条件
LD TR0
AND 505.08  ; 0条件
ANDNOT 822.14  ; #1-2电池抽真空阀开到位标志
AND 823.03  ; #1-2电池注氦阀关到位标志
AND 823.07  ; #1-2电池破真空阀关到位标志
ANDNOT 515.08  ; 条件
OUT 605.08  ; #1-2电池氦气回收阀开[A]
LD TR0
AND 515.08  ; 条件
ANDNOT 822.15  ; #1-2电池抽真空阀关到位标志
ANDNOT 505.08  ; 0条件
OUT 615.08  ; #1-2电池氦气回收阀关[A]

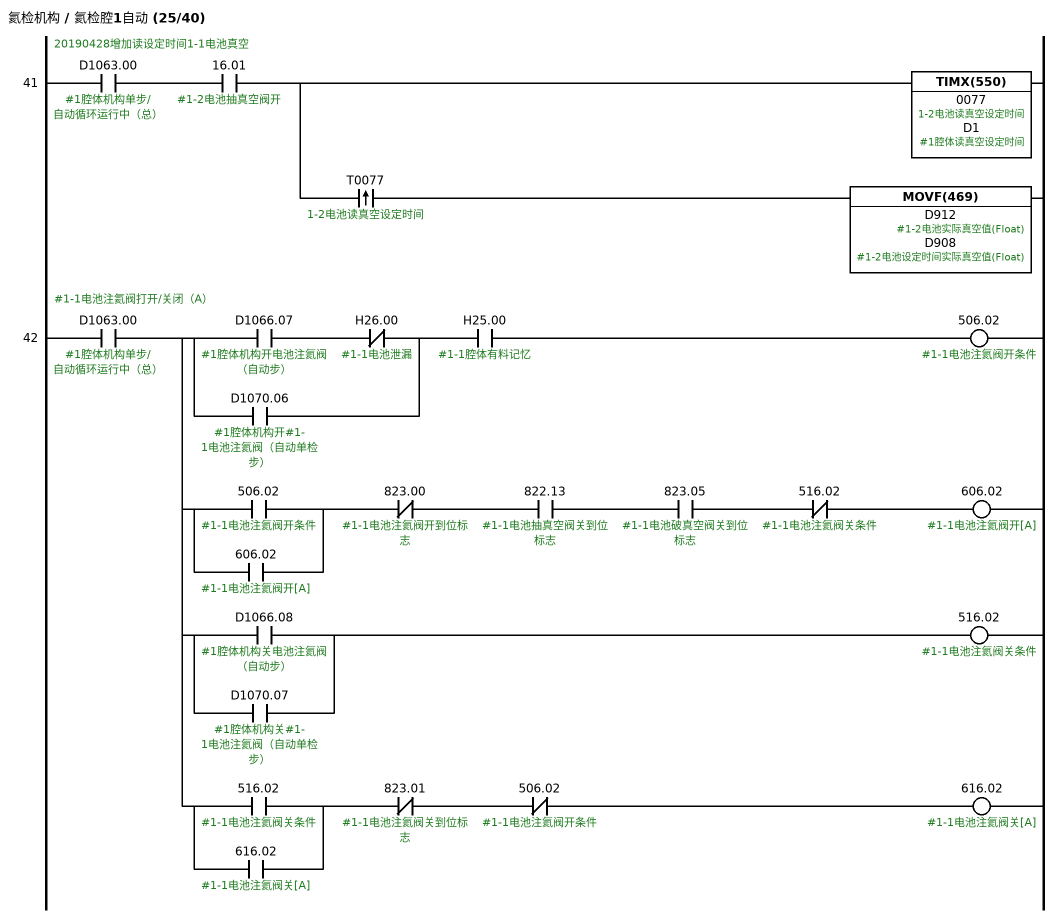
; rung 41: 20190428增加读设定时间1-1电池真空
LD D1063.00  ; #1腔体机构单步/自动循环运行中（总）
AND 16.01  ; #1-2电池抽真空阀开
TIMX(550) 0077 D1  ; #1腔体读真空设定时间, 1-2电池读真空设定时间
@AND T0077  ; 1-2电池读真空设定时间
MOVF(469) D912 D908  ; #1-2电池实际真空值(Float), #1-2电池设定时间实际真空值(Float)
; rung 42: #1-1电池注氦阀打开/关闭（A）
LD D1063.00  ; #1腔体机构单步/自动循环运行中（总）
OUT TR0
LD D1066.07  ; #1腔体机构开电池注氦阀（自动步）
ANDNOT H26.00  ; #1-1电池泄漏
OR D1070.06  ; #1腔体机构开#1-1电池注氦阀（自动单检步）
ANDLD
AND H25.00  ; #1-1腔体有料记忆
OUT 506.02  ; #1-1电池注氦阀开条件
LD TR0
LD 506.02  ; #1-1电池注氦阀开条件
OR 606.02  ; #1-1电池注氦阀开[A]
ANDLD
ANDNOT 823.00  ; #1-1电池注氦阀开到位标志
AND 822.13  ; #1-1电池抽真空阀关到位标志
AND 823.05  ; #1-1电池破真空阀关到位标志
ANDNOT 516.02  ; #1-1电池注氦阀关条件
OUT 606.02  ; #1-1电池注氦阀开[A]
LD TR0
LD D1066.08  ; #1腔体机构关电池注氦阀（自动步）
OR D1070.07  ; #1腔体机构关#1-1电池注氦阀（自动单检步）
ANDLD
OUT 516.02  ; #1-1电池注氦阀关条件
LD TR0
LD 516.02  ; #1-1电池注氦阀关条件
OR 616.02  ; #1-1电池注氦阀关[A]
ANDLD
ANDNOT 823.01  ; #1-1电池注氦阀关到位标志
ANDNOT 506.02  ; #1-1电池注氦阀开条件
OUT 616.02  ; #1-1电池注氦阀关[A]

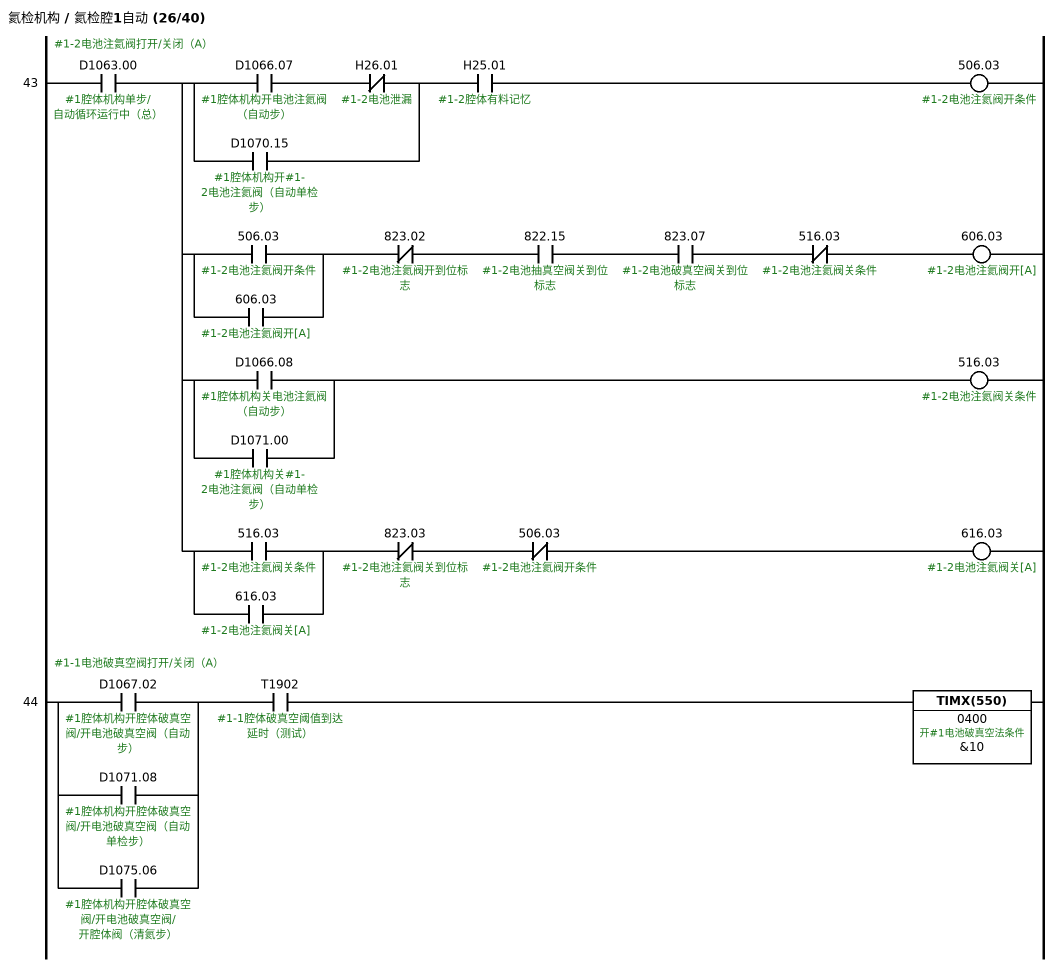
; rung 43: #1-2电池注氦阀打开/关闭（A）
LD D1063.00  ; #1腔体机构单步/自动循环运行中（总）
OUT TR0
LD D1066.07  ; #1腔体机构开电池注氦阀（自动步）
ANDNOT H26.01  ; #1-2电池泄漏
OR D1070.15  ; #1腔体机构开#1-2电池注氦阀（自动单检步）
ANDLD
AND H25.01  ; #1-2腔体有料记忆
OUT 506.03  ; #1-2电池注氦阀开条件
LD TR0
LD 506.03  ; #1-2电池注氦阀开条件
OR 606.03  ; #1-2电池注氦阀开[A]
ANDLD
ANDNOT 823.02  ; #1-2电池注氦阀开到位标志
AND 822.15  ; #1-2电池抽真空阀关到位标志
AND 823.07  ; #1-2电池破真空阀关到位标志
ANDNOT 516.03  ; #1-2电池注氦阀关条件
OUT 606.03  ; #1-2电池注氦阀开[A]
LD TR0
LD D1066.08  ; #1腔体机构关电池注氦阀（自动步）
OR D1071.00  ; #1腔体机构关#1-2电池注氦阀（自动单检步）
ANDLD
OUT 516.03  ; #1-2电池注氦阀关条件
LD TR0
LD 516.03  ; #1-2电池注氦阀关条件
OR 616.03  ; #1-2电池注氦阀关[A]
ANDLD
ANDNOT 823.03  ; #1-2电池注氦阀关到位标志
ANDNOT 506.03  ; #1-2电池注氦阀开条件
OUT 616.03  ; #1-2电池注氦阀关[A]
; rung 44: #1-1电池破真空阀打开/关闭（A）
LD D1067.02  ; #1腔体机构开腔体破真空阀/开电池破真空阀（自动步）
OR D1071.08  ; #1腔体机构开腔体破真空阀/开电池破真空阀（自动单检步）
OR D1075.06  ; #1腔体机构开腔体破真空阀/开电池破真空阀/开腔体阀（清氦步）
AND T1902  ; #1-1腔体破真空阈值到达延时（测试）
TIMX(550) 0400 &10  ; 开#1电池破真空法条件

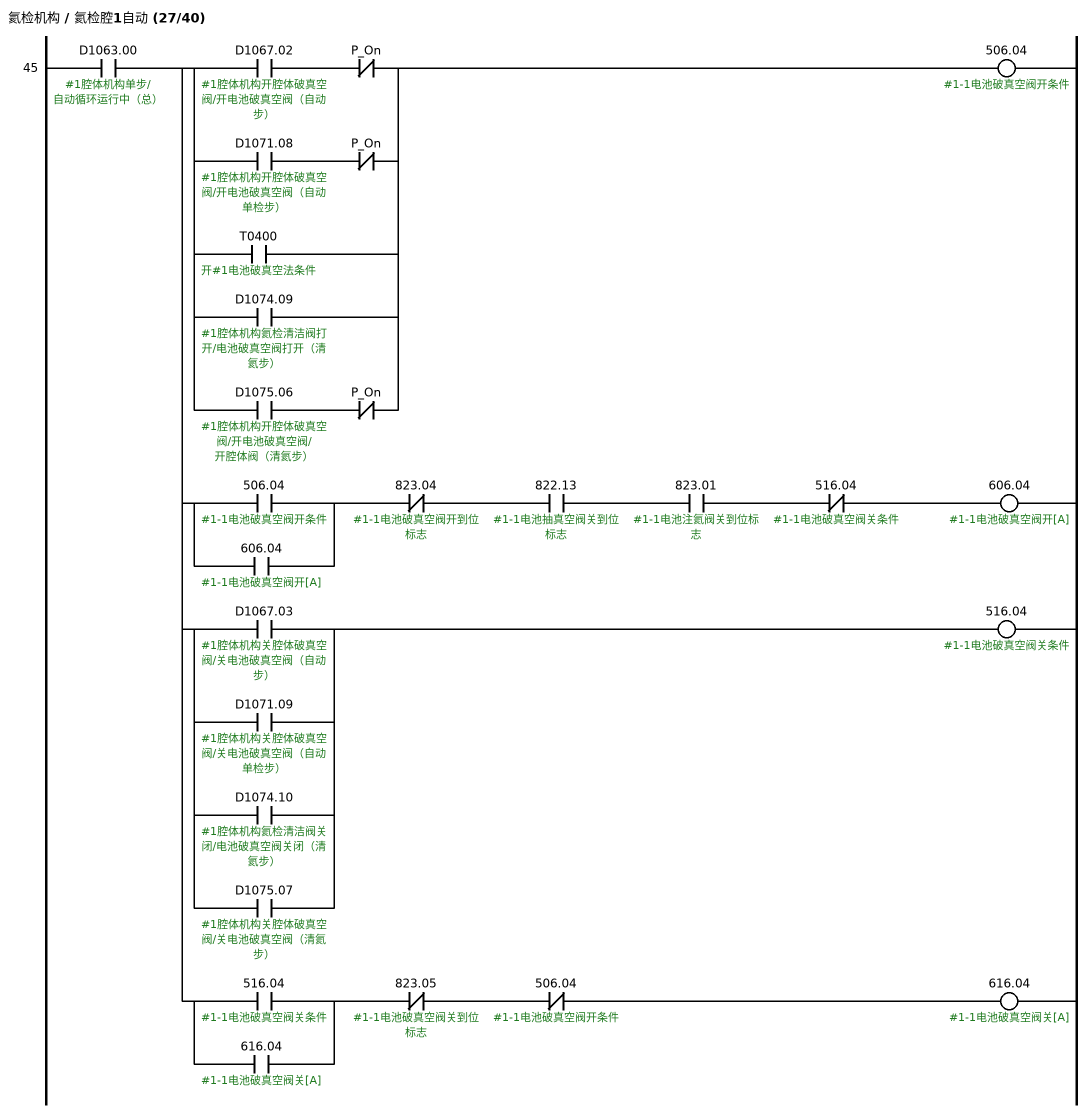
; rung 45
LD D1063.00  ; #1腔体机构单步/自动循环运行中（总）
OUT TR0
LD D1067.02  ; #1腔体机构开腔体破真空阀/开电池破真空阀（自动步）
ANDNOT P_On
LD D1071.08  ; #1腔体机构开腔体破真空阀/开电池破真空阀（自动单检步）
ANDNOT P_On
ORLD
OR T0400  ; 开#1电池破真空法条件
OR D1074.09  ; #1腔体机构氦检清洁阀打开/电池破真空阀打开（清氦步）
LD D1075.06  ; #1腔体机构开腔体破真空阀/开电池破真空阀/开腔体阀（清氦步）
ANDNOT P_On
ORLD
ANDLD
OUT 506.04  ; #1-1电池破真空阀开条件
LD TR0
LD 506.04  ; #1-1电池破真空阀开条件
OR 606.04  ; #1-1电池破真空阀开[A]
ANDLD
ANDNOT 823.04  ; #1-1电池破真空阀开到位标志
AND 822.13  ; #1-1电池抽真空阀关到位标志
AND 823.01  ; #1-1电池注氦阀关到位标志
ANDNOT 516.04  ; #1-1电池破真空阀关条件
OUT 606.04  ; #1-1电池破真空阀开[A]
LD TR0
LD D1067.03  ; #1腔体机构关腔体破真空阀/关电池破真空阀（自动步）
OR D1071.09  ; #1腔体机构关腔体破真空阀/关电池破真空阀（自动单检步）
OR D1074.10  ; #1腔体机构氦检清洁阀关闭/电池破真空阀关闭（清氦步）
OR D1075.07  ; #1腔体机构关腔体破真空阀/关电池破真空阀（清氦步）
ANDLD
OUT 516.04  ; #1-1电池破真空阀关条件
LD TR0
LD 516.04  ; #1-1电池破真空阀关条件
OR 616.04  ; #1-1电池破真空阀关[A]
ANDLD
ANDNOT 823.05  ; #1-1电池破真空阀关到位标志
ANDNOT 506.04  ; #1-1电池破真空阀开条件
OUT 616.04  ; #1-1电池破真空阀关[A]

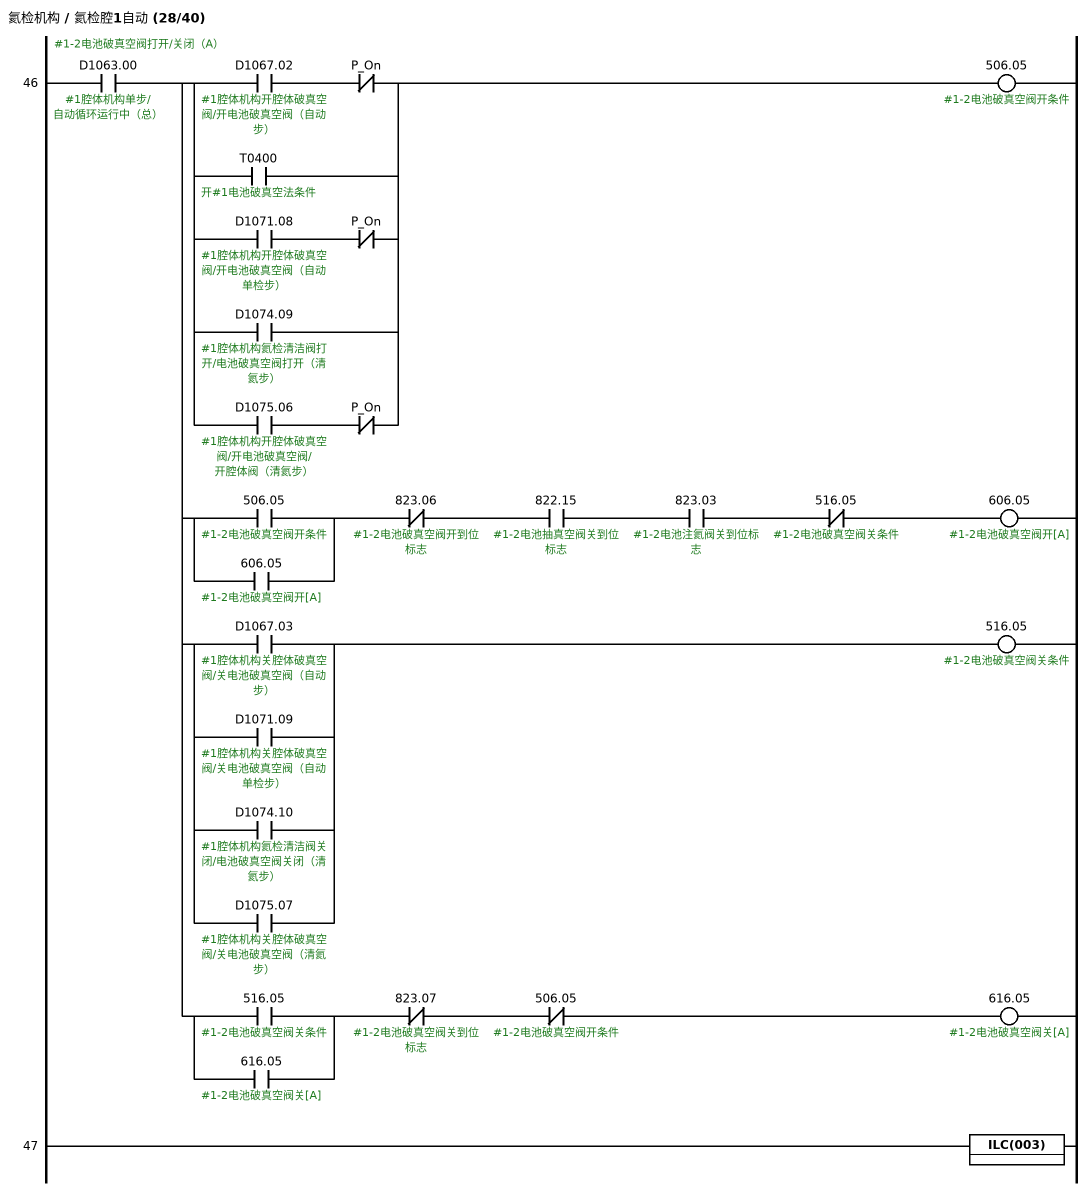
; rung 46: #1-2电池破真空阀打开/关闭（A）
LD D1063.00  ; #1腔体机构单步/自动循环运行中（总）
OUT TR0
LD D1067.02  ; #1腔体机构开腔体破真空阀/开电池破真空阀（自动步）
ANDNOT P_On
OR T0400  ; 开#1电池破真空法条件
LD D1071.08  ; #1腔体机构开腔体破真空阀/开电池破真空阀（自动单检步）
ANDNOT P_On
ORLD
OR D1074.09  ; #1腔体机构氦检清洁阀打开/电池破真空阀打开（清氦步）
LD D1075.06  ; #1腔体机构开腔体破真空阀/开电池破真空阀/开腔体阀（清氦步）
ANDNOT P_On
ORLD
ANDLD
OUT 506.05  ; #1-2电池破真空阀开条件
LD TR0
LD 506.05  ; #1-2电池破真空阀开条件
OR 606.05  ; #1-2电池破真空阀开[A]
ANDLD
ANDNOT 823.06  ; #1-2电池破真空阀开到位标志
AND 822.15  ; #1-2电池抽真空阀关到位标志
AND 823.03  ; #1-2电池注氦阀关到位标志
ANDNOT 516.05  ; #1-2电池破真空阀关条件
OUT 606.05  ; #1-2电池破真空阀开[A]
LD TR0
LD D1067.03  ; #1腔体机构关腔体破真空阀/关电池破真空阀（自动步）
OR D1071.09  ; #1腔体机构关腔体破真空阀/关电池破真空阀（自动单检步）
OR D1074.10  ; #1腔体机构氦检清洁阀关闭/电池破真空阀关闭（清氦步）
OR D1075.07  ; #1腔体机构关腔体破真空阀/关电池破真空阀（清氦步）
ANDLD
OUT 516.05  ; #1-2电池破真空阀关条件
LD TR0
LD 516.05  ; #1-2电池破真空阀关条件
OR 616.05  ; #1-2电池破真空阀关[A]
ANDLD
ANDNOT 823.07  ; #1-2电池破真空阀关到位标志
ANDNOT 506.05  ; #1-2电池破真空阀开条件
OUT 616.05  ; #1-2电池破真空阀关[A]
; rung 47
ILC(003)

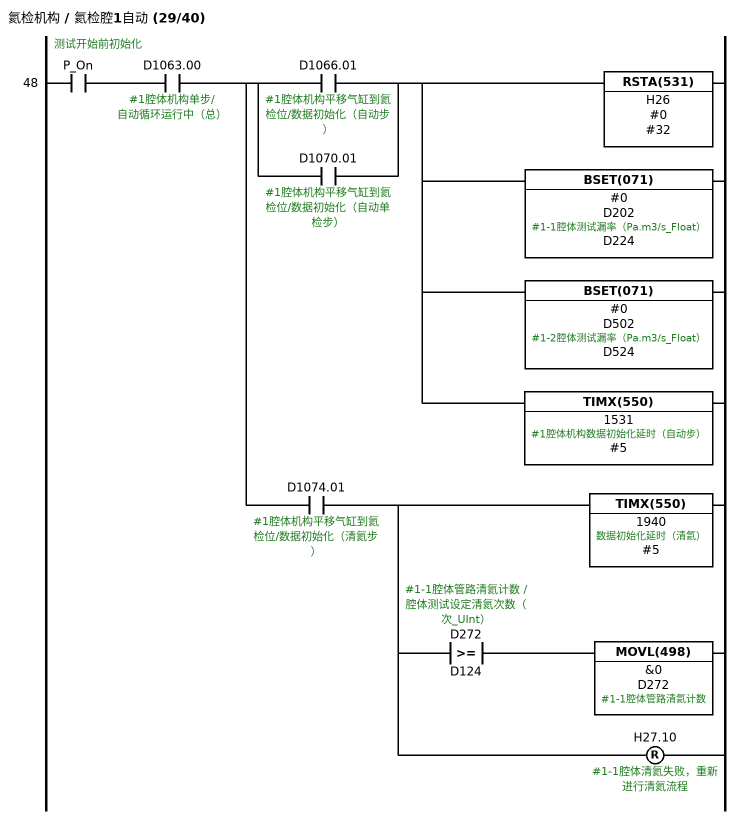
; rung 48: 测试开始前初始化
LD P_On
AND D1063.00  ; #1腔体机构单步/自动循环运行中（总）
OUT TR0
LD D1066.01  ; #1腔体机构平移气缸到氦检位/数据初始化（自动步）
OR D1070.01  ; #1腔体机构平移气缸到氦检位/数据初始化（自动单检步）
ANDLD
RSTA(531) H26 #0 #32
BSET(071) #0 D202 D224  ; #1-1腔体测试漏率（Pa.m3/s_Float）
BSET(071) #0 D502 D524  ; #1-2腔体测试漏率（Pa.m3/s_Float）
TIMX(550) 1531 #5  ; #1腔体机构数据初始化延时（自动步）
LD TR0
AND D1074.01  ; #1腔体机构平移气缸到氦检位/数据初始化（清氦步）
OUT TR0
TIMX(550) 1940 #5  ; 数据初始化延时（清氦）
AND>=(325) D272 D124  ; #1-1腔体管路清氦计数, 腔体测试设定清氦次数（次_UInt）
MOVL(498) &0 D272  ; #1-1腔体管路清氦计数
LD TR0
RSET H27.10  ; #1-1腔体清氦失败，重新进行清氦流程

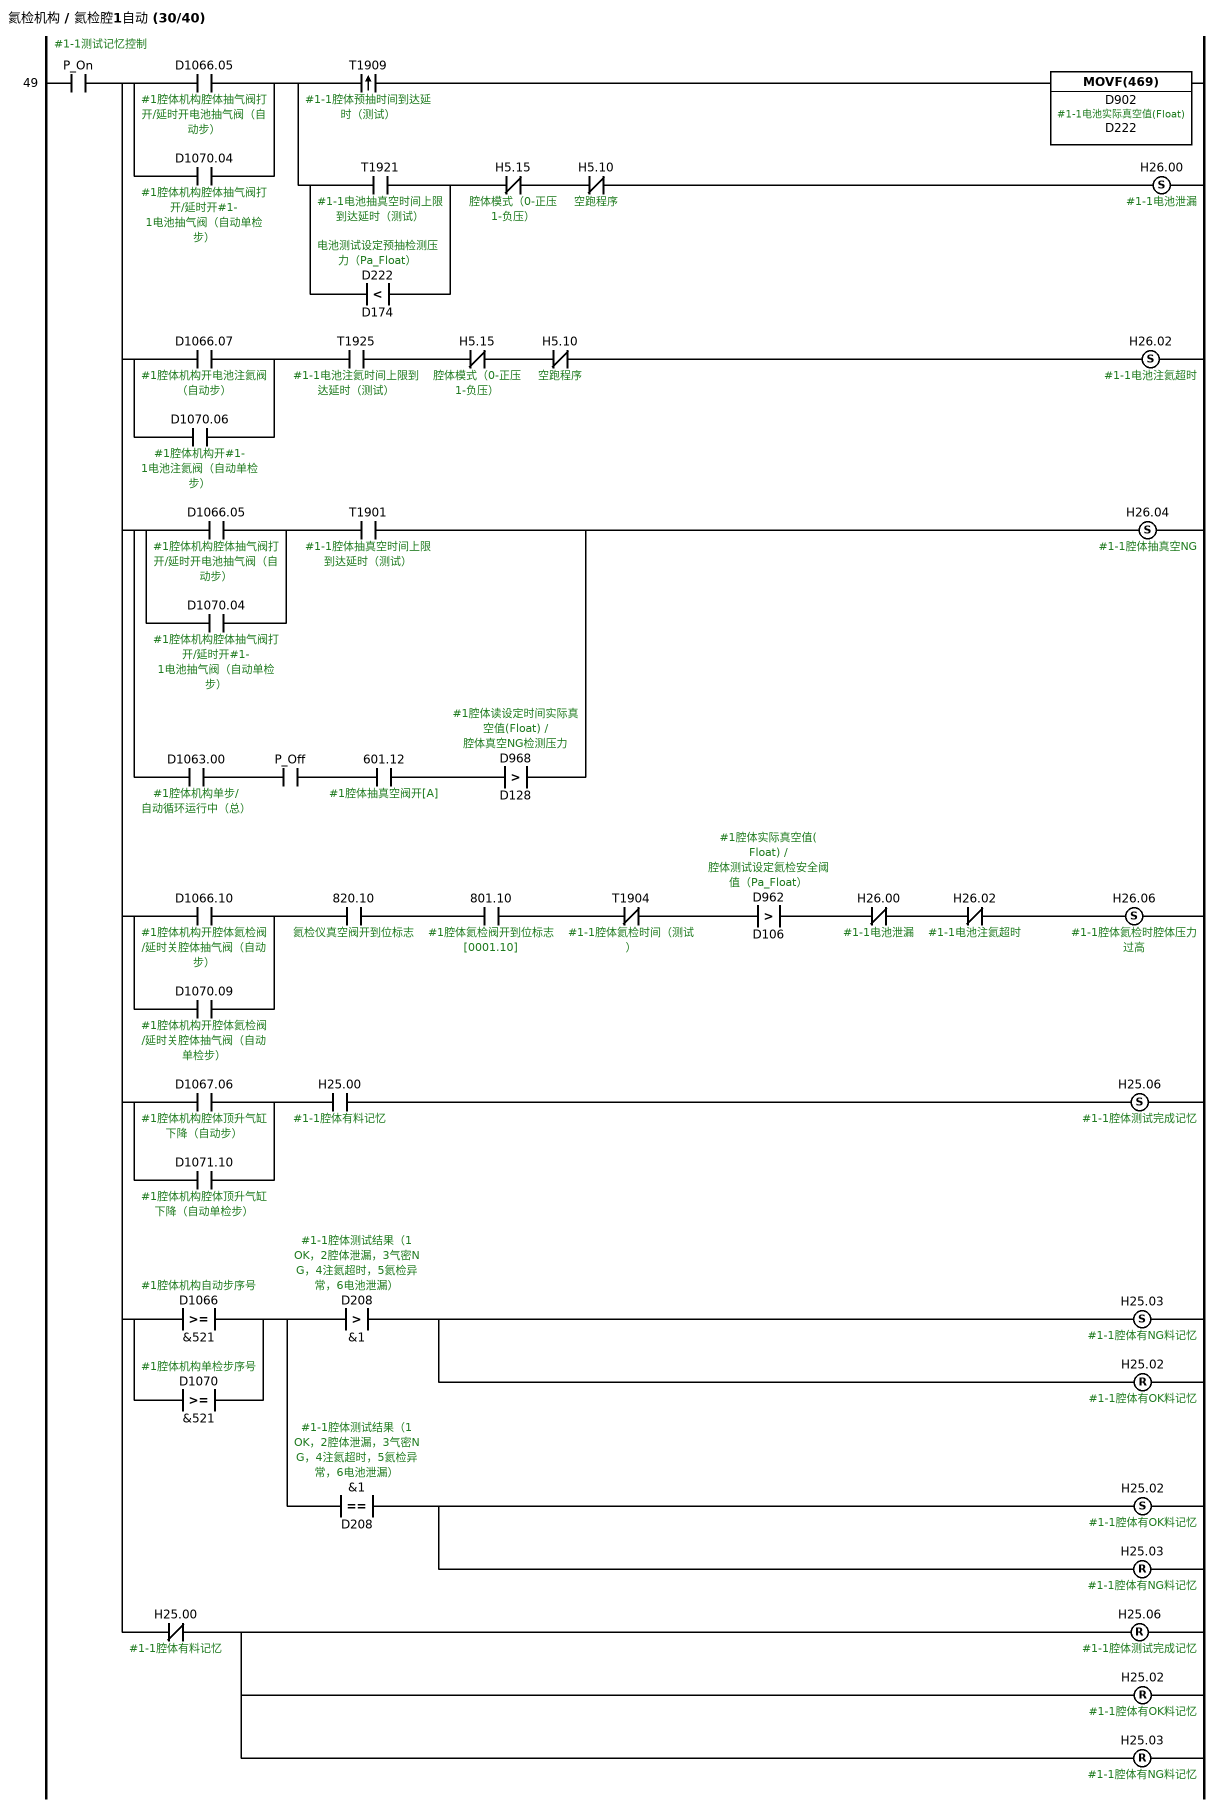
; rung 49: #1-1测试记忆控制
LD P_On
OUT TR0
LD D1066.05  ; #1腔体机构腔体抽气阀打开/延时开电池抽气阀（自动步）
OR D1070.04  ; #1腔体机构腔体抽气阀打开/延时开#1-1电池抽气阀（自动单检步）
ANDLD
OUT TR1
@AND T1909  ; #1-1腔体预抽时间到达延时（测试）
MOVF(469) D902 D222  ; #1-1电池实际真空值(Float)
LD TR1
LD T1921  ; #1-1电池抽真空时间上限到达延时（测试）
OR<F(331) D222 D174  ; 电池测试设定预抽检测压力（Pa_Float）
ANDLD
ANDNOT H5.15  ; 腔体模式（0-正压 1-负压）
ANDNOT H5.10  ; 空跑程序
SET H26.00  ; #1-1电池泄漏
LD TR0
LD D1066.07  ; #1腔体机构开电池注氦阀（自动步）
OR D1070.06  ; #1腔体机构开#1-1电池注氦阀（自动单检步）
ANDLD
AND T1925  ; #1-1电池注氦时间上限到达延时（测试）
ANDNOT H5.15  ; 腔体模式（0-正压 1-负压）
ANDNOT H5.10  ; 空跑程序
SET H26.02  ; #1-1电池注氦超时
LD TR0
LD D1066.05  ; #1腔体机构腔体抽气阀打开/延时开电池抽气阀（自动步）
OR D1070.04  ; #1腔体机构腔体抽气阀打开/延时开#1-1电池抽气阀（自动单检步）
AND T1901  ; #1-1腔体抽真空时间上限到达延时（测试）
LD D1063.00  ; #1腔体机构单步/自动循环运行中（总）
AND P_Off
AND 601.12  ; #1腔体抽真空阀开[A]
AND>F(333) D968 D128  ; #1腔体读设定时间实际真空值(Float), 腔体真空NG检测压力
ORLD
ANDLD
SET H26.04  ; #1-1腔体抽真空NG
LD TR0
LD D1066.10  ; #1腔体机构开腔体氦检阀/延时关腔体抽气阀（自动步）
OR D1070.09  ; #1腔体机构开腔体氦检阀/延时关腔体抽气阀（自动单检步）
ANDLD
AND 820.10  ; 氦检仪真空阀开到位标志
AND 801.10  ; #1腔体氦检阀开到位标志[0001.10]
ANDNOT T1904  ; #1-1腔体氦检时间（测试）
AND>F(333) D962 D106  ; #1腔体实际真空值(Float), 腔体测试设定氦检安全阈值（Pa_Float）
ANDNOT H26.00  ; #1-1电池泄漏
ANDNOT H26.02  ; #1-1电池注氦超时
SET H26.06  ; #1-1腔体氦检时腔体压力过高
LD TR0
LD D1067.06  ; #1腔体机构腔体顶升气缸下降（自动步）
OR D1071.10  ; #1腔体机构腔体顶升气缸下降（自动单检步）
ANDLD
AND H25.00  ; #1-1腔体有料记忆
SET H25.06  ; #1-1腔体测试完成记忆
LD TR0
LD>=L(326) D1066 &521  ; #1腔体机构自动步序号
OR>=L(326) D1070 &521  ; #1腔体机构单检步序号
ANDLD
OUT TR1
AND>(320) D208 &1  ; #1-1腔体测试结果（1 OK，2腔体泄漏，3气密NG，4注氦超时，5氦检异常，6电池泄漏）
SET H25.03  ; #1-1腔体有NG料记忆
RSET H25.02  ; #1-1腔体有OK料记忆
LD TR1
AND=(300) &1 D208  ; #1-1腔体测试结果（1 OK，2腔体泄漏，3气密NG，4注氦超时，5氦检异常，6电池泄漏）
SET H25.02  ; #1-1腔体有OK料记忆
RSET H25.03  ; #1-1腔体有NG料记忆
LD TR0
ANDNOT H25.00  ; #1-1腔体有料记忆
RSET H25.06  ; #1-1腔体测试完成记忆
RSET H25.02  ; #1-1腔体有OK料记忆
RSET H25.03  ; #1-1腔体有NG料记忆

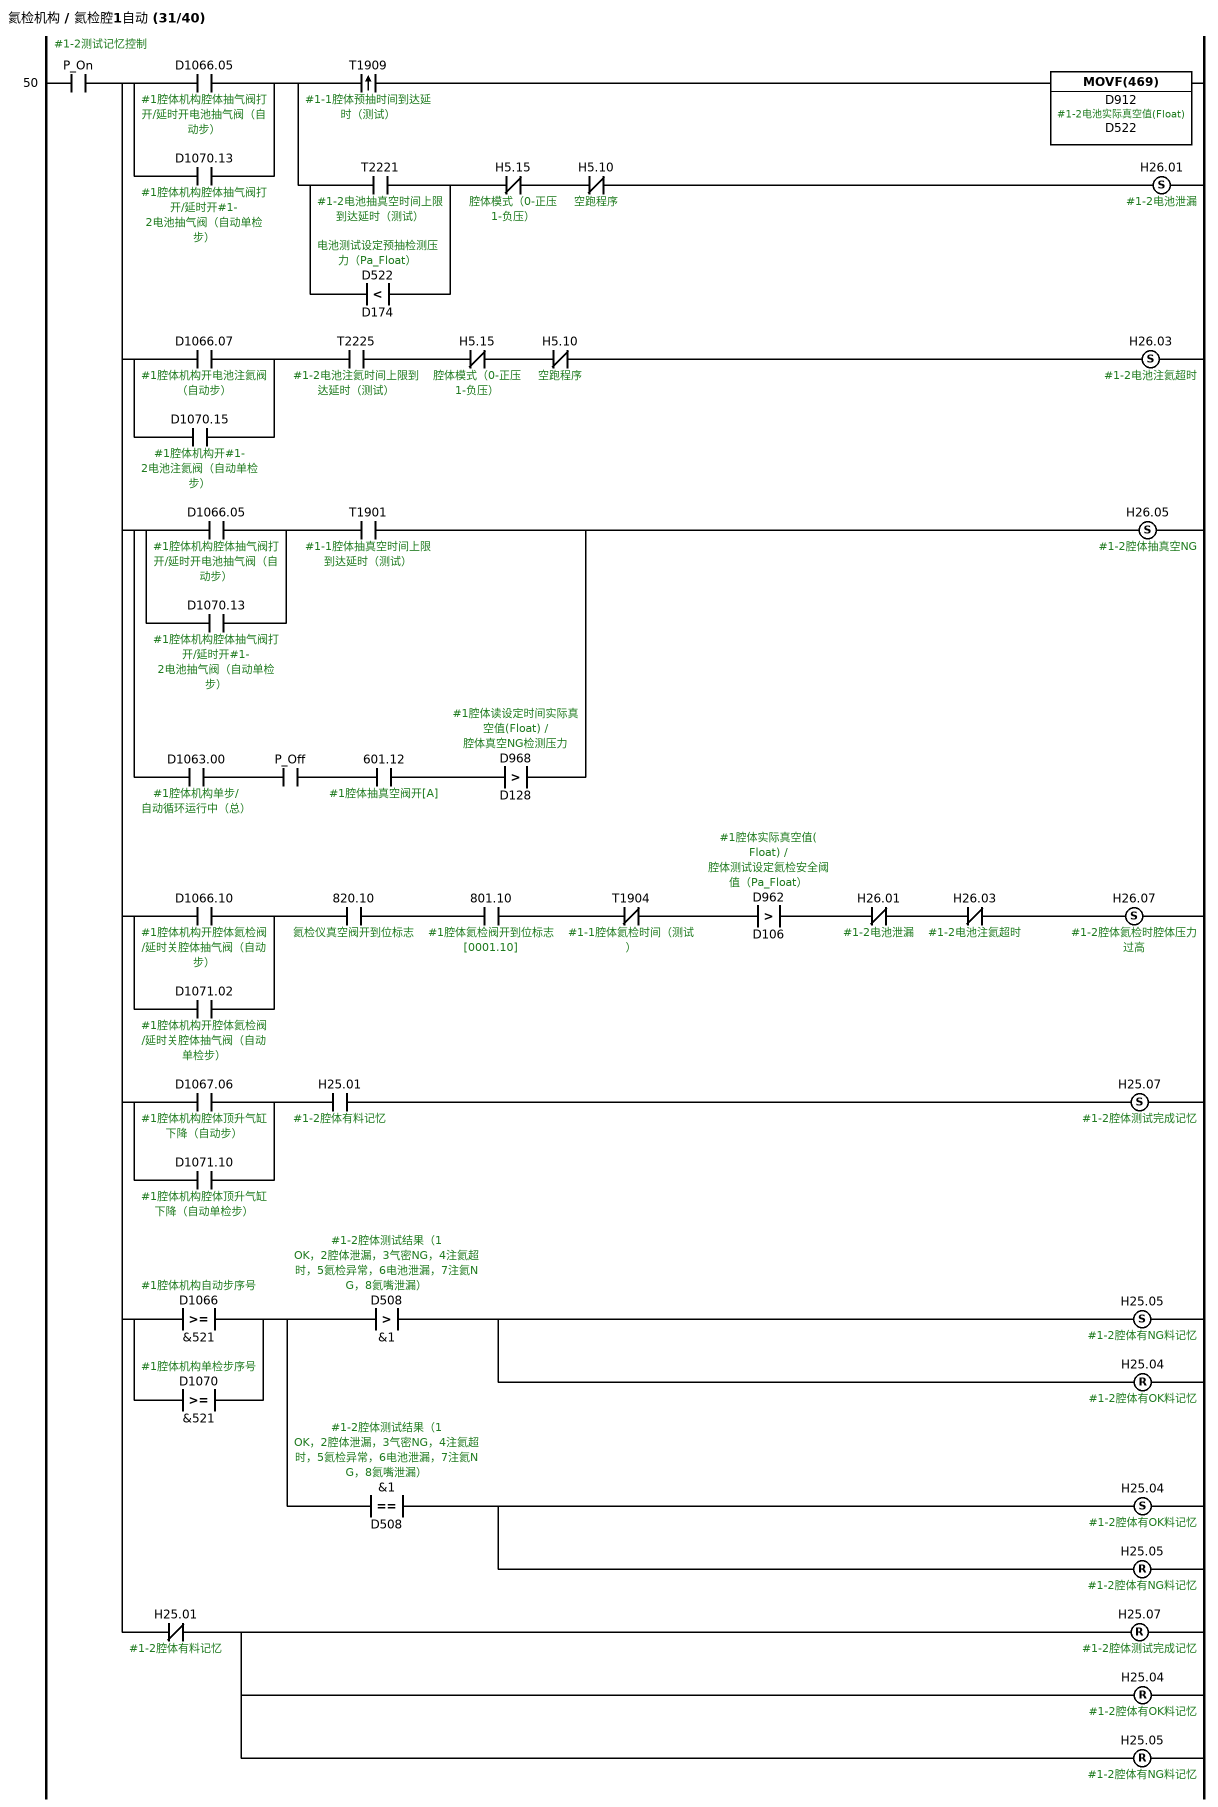
; rung 50: #1-2测试记忆控制
LD P_On
OUT TR0
LD D1066.05  ; #1腔体机构腔体抽气阀打开/延时开电池抽气阀（自动步）
OR D1070.13  ; #1腔体机构腔体抽气阀打开/延时开#1-2电池抽气阀（自动单检步）
ANDLD
OUT TR1
@AND T1909  ; #1-1腔体预抽时间到达延时（测试）
MOVF(469) D912 D522  ; #1-2电池实际真空值(Float)
LD TR1
LD T2221  ; #1-2电池抽真空时间上限到达延时（测试）
OR<F(331) D522 D174  ; 电池测试设定预抽检测压力（Pa_Float）
ANDLD
ANDNOT H5.15  ; 腔体模式（0-正压 1-负压）
ANDNOT H5.10  ; 空跑程序
SET H26.01  ; #1-2电池泄漏
LD TR0
LD D1066.07  ; #1腔体机构开电池注氦阀（自动步）
OR D1070.15  ; #1腔体机构开#1-2电池注氦阀（自动单检步）
ANDLD
AND T2225  ; #1-2电池注氦时间上限到达延时（测试）
ANDNOT H5.15  ; 腔体模式（0-正压 1-负压）
ANDNOT H5.10  ; 空跑程序
SET H26.03  ; #1-2电池注氦超时
LD TR0
LD D1066.05  ; #1腔体机构腔体抽气阀打开/延时开电池抽气阀（自动步）
OR D1070.13  ; #1腔体机构腔体抽气阀打开/延时开#1-2电池抽气阀（自动单检步）
AND T1901  ; #1-1腔体抽真空时间上限到达延时（测试）
LD D1063.00  ; #1腔体机构单步/自动循环运行中（总）
AND P_Off
AND 601.12  ; #1腔体抽真空阀开[A]
AND>F(333) D968 D128  ; #1腔体读设定时间实际真空值(Float), 腔体真空NG检测压力
ORLD
ANDLD
SET H26.05  ; #1-2腔体抽真空NG
LD TR0
LD D1066.10  ; #1腔体机构开腔体氦检阀/延时关腔体抽气阀（自动步）
OR D1071.02  ; #1腔体机构开腔体氦检阀/延时关腔体抽气阀（自动单检步）
ANDLD
AND 820.10  ; 氦检仪真空阀开到位标志
AND 801.10  ; #1腔体氦检阀开到位标志[0001.10]
ANDNOT T1904  ; #1-1腔体氦检时间（测试）
AND>F(333) D962 D106  ; #1腔体实际真空值(Float), 腔体测试设定氦检安全阈值（Pa_Float）
ANDNOT H26.01  ; #1-2电池泄漏
ANDNOT H26.03  ; #1-2电池注氦超时
SET H26.07  ; #1-2腔体氦检时腔体压力过高
LD TR0
LD D1067.06  ; #1腔体机构腔体顶升气缸下降（自动步）
OR D1071.10  ; #1腔体机构腔体顶升气缸下降（自动单检步）
ANDLD
AND H25.01  ; #1-2腔体有料记忆
SET H25.07  ; #1-2腔体测试完成记忆
LD TR0
LD>=L(326) D1066 &521  ; #1腔体机构自动步序号
OR>=L(326) D1070 &521  ; #1腔体机构单检步序号
ANDLD
OUT TR1
AND>(320) D508 &1  ; #1-2腔体测试结果（1 OK，2腔体泄漏，3气密NG，4注氦超时，5氦检异常，6电池泄漏，7注氦NG，8氦嘴泄漏）
SET H25.05  ; #1-2腔体有NG料记忆
RSET H25.04  ; #1-2腔体有OK料记忆
LD TR1
AND=(300) &1 D508  ; #1-2腔体测试结果（1 OK，2腔体泄漏，3气密NG，4注氦超时，5氦检异常，6电池泄漏，7注氦NG，8氦嘴泄漏）
SET H25.04  ; #1-2腔体有OK料记忆
RSET H25.05  ; #1-2腔体有NG料记忆
LD TR0
ANDNOT H25.01  ; #1-2腔体有料记忆
RSET H25.07  ; #1-2腔体测试完成记忆
RSET H25.04  ; #1-2腔体有OK料记忆
RSET H25.05  ; #1-2腔体有NG料记忆

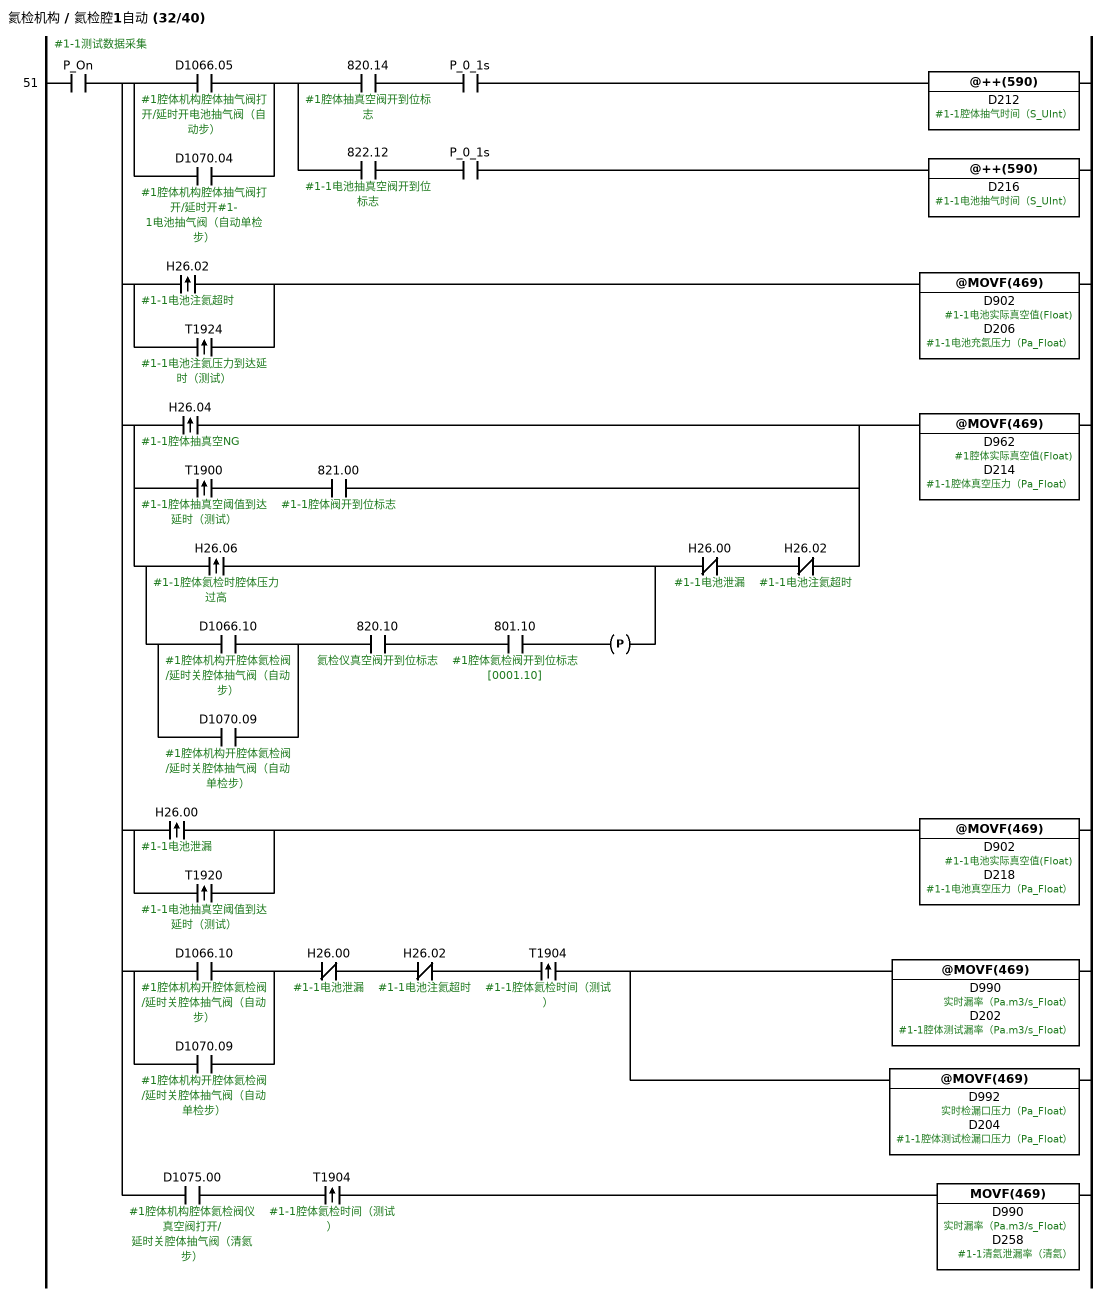
; rung 51: #1-1测试数据采集
LD P_On
OUT TR0
LD D1066.05  ; #1腔体机构腔体抽气阀打开/延时开电池抽气阀（自动步）
OR D1070.04  ; #1腔体机构腔体抽气阀打开/延时开#1-1电池抽气阀（自动单检步）
ANDLD
OUT TR1
AND 820.14  ; #1腔体抽真空阀开到位标志
AND P_0_1s
@++(590) D212  ; #1-1腔体抽气时间（S_UInt）
LD TR1
AND 822.12  ; #1-1电池抽真空阀开到位标志
AND P_0_1s
@++(590) D216  ; #1-1电池抽气时间（S_UInt）
LD TR0
@LD H26.02  ; #1-1电池注氦超时
@OR T1924  ; #1-1电池注氦压力到达延时（测试）
ANDLD
@MOVF(469) D902 D206  ; #1-1电池实际真空值(Float), #1-1电池充氦压力（Pa_Float）
LD TR0
@LD H26.04  ; #1-1腔体抽真空NG
@LD T1900  ; #1-1腔体抽真空阈值到达延时（测试）
AND 821.00  ; #1-1腔体阀开到位标志
ORLD
@LD H26.06  ; #1-1腔体氦检时腔体压力过高
LD D1066.10  ; #1腔体机构开腔体氦检阀/延时关腔体抽气阀（自动步）
OR D1070.09  ; #1腔体机构开腔体氦检阀/延时关腔体抽气阀（自动单检步）
AND 820.10  ; 氦检仪真空阀开到位标志
AND 801.10  ; #1腔体氦检阀开到位标志[0001.10]
UP(521)
ORLD
ANDNOT H26.00  ; #1-1电池泄漏
ANDNOT H26.02  ; #1-1电池注氦超时
ORLD
ANDLD
@MOVF(469) D962 D214  ; #1腔体实际真空值(Float), #1-1腔体真空压力（Pa_Float）
LD TR0
@LD H26.00  ; #1-1电池泄漏
@OR T1920  ; #1-1电池抽真空阈值到达延时（测试）
ANDLD
@MOVF(469) D902 D218  ; #1-1电池实际真空值(Float), #1-1电池真空压力（Pa_Float）
LD TR0
LD D1066.10  ; #1腔体机构开腔体氦检阀/延时关腔体抽气阀（自动步）
OR D1070.09  ; #1腔体机构开腔体氦检阀/延时关腔体抽气阀（自动单检步）
ANDLD
ANDNOT H26.00  ; #1-1电池泄漏
ANDNOT H26.02  ; #1-1电池注氦超时
@AND T1904  ; #1-1腔体氦检时间（测试）
@MOVF(469) D990 D202  ; 实时漏率（Pa.m3/s_Float）, #1-1腔体测试漏率（Pa.m3/s_Float）
@MOVF(469) D992 D204  ; 实时检漏口压力（Pa_Float）, #1-1腔体测试检漏口压力（Pa_Float）
LD TR0
AND D1075.00  ; #1腔体机构腔体氦检阀仪真空阀打开/延时关腔体抽气阀（清氦步）
@AND T1904  ; #1-1腔体氦检时间（测试）
MOVF(469) D990 D258  ; 实时漏率（Pa.m3/s_Float）, #1-1清氦泄漏率（清氦）

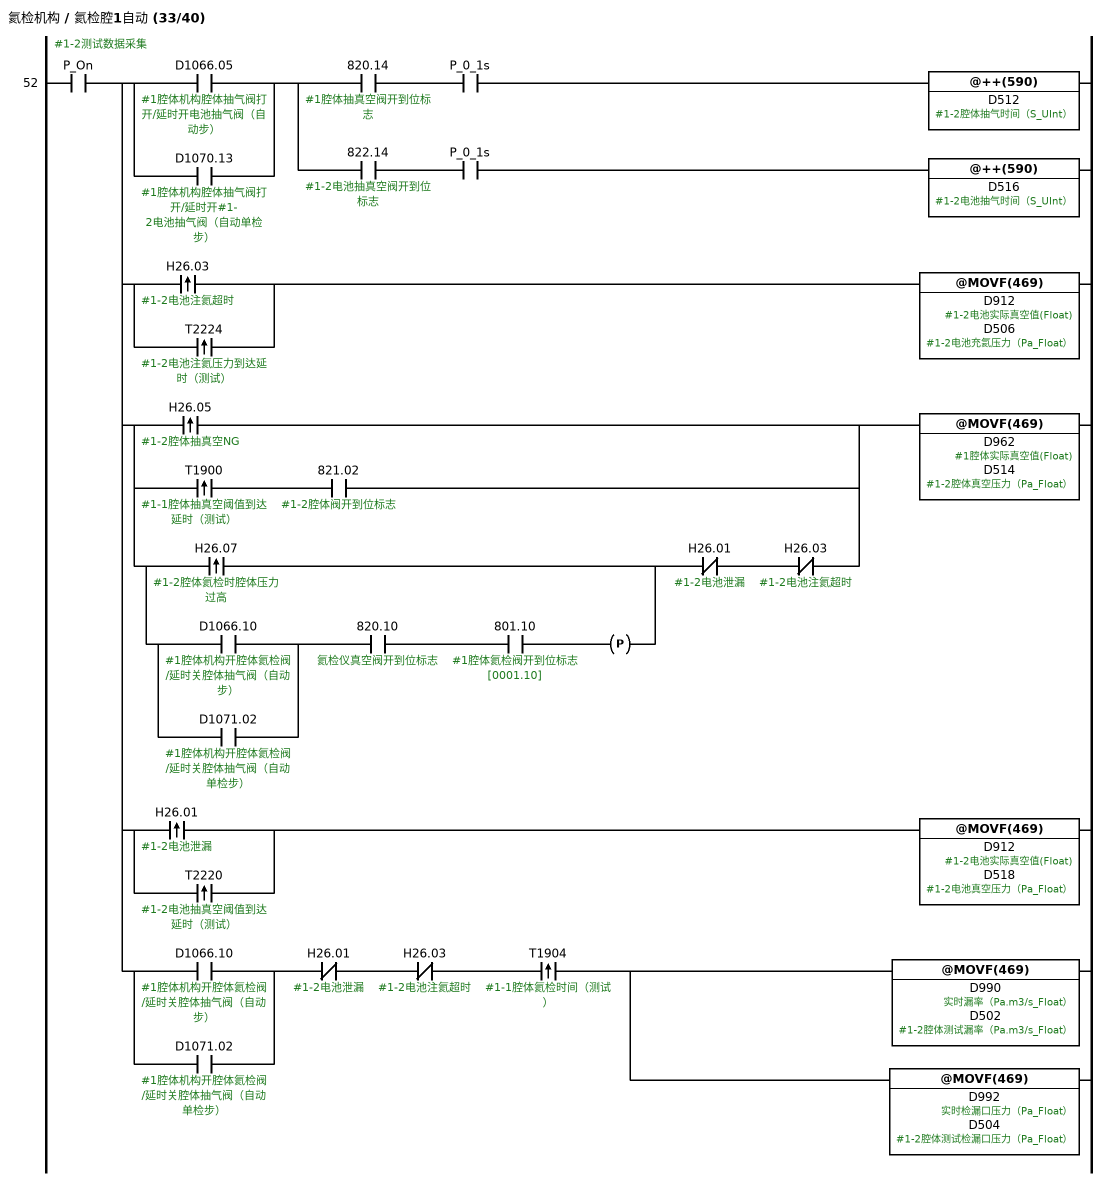
; rung 52: #1-2测试数据采集
LD P_On
OUT TR0
LD D1066.05  ; #1腔体机构腔体抽气阀打开/延时开电池抽气阀（自动步）
OR D1070.13  ; #1腔体机构腔体抽气阀打开/延时开#1-2电池抽气阀（自动单检步）
ANDLD
OUT TR1
AND 820.14  ; #1腔体抽真空阀开到位标志
AND P_0_1s
@++(590) D512  ; #1-2腔体抽气时间（S_UInt）
LD TR1
AND 822.14  ; #1-2电池抽真空阀开到位标志
AND P_0_1s
@++(590) D516  ; #1-2电池抽气时间（S_UInt）
LD TR0
@LD H26.03  ; #1-2电池注氦超时
@OR T2224  ; #1-2电池注氦压力到达延时（测试）
ANDLD
@MOVF(469) D912 D506  ; #1-2电池实际真空值(Float), #1-2电池充氦压力（Pa_Float）
LD TR0
@LD H26.05  ; #1-2腔体抽真空NG
@LD T1900  ; #1-1腔体抽真空阈值到达延时（测试）
AND 821.02  ; #1-2腔体阀开到位标志
ORLD
@LD H26.07  ; #1-2腔体氦检时腔体压力过高
LD D1066.10  ; #1腔体机构开腔体氦检阀/延时关腔体抽气阀（自动步）
OR D1071.02  ; #1腔体机构开腔体氦检阀/延时关腔体抽气阀（自动单检步）
AND 820.10  ; 氦检仪真空阀开到位标志
AND 801.10  ; #1腔体氦检阀开到位标志[0001.10]
UP(521)
ORLD
ANDNOT H26.01  ; #1-2电池泄漏
ANDNOT H26.03  ; #1-2电池注氦超时
ORLD
ANDLD
@MOVF(469) D962 D514  ; #1腔体实际真空值(Float), #1-2腔体真空压力（Pa_Float）
LD TR0
@LD H26.01  ; #1-2电池泄漏
@OR T2220  ; #1-2电池抽真空阈值到达延时（测试）
ANDLD
@MOVF(469) D912 D518  ; #1-2电池实际真空值(Float), #1-2电池真空压力（Pa_Float）
LD TR0
LD D1066.10  ; #1腔体机构开腔体氦检阀/延时关腔体抽气阀（自动步）
OR D1071.02  ; #1腔体机构开腔体氦检阀/延时关腔体抽气阀（自动单检步）
ANDLD
ANDNOT H26.01  ; #1-2电池泄漏
ANDNOT H26.03  ; #1-2电池注氦超时
@AND T1904  ; #1-1腔体氦检时间（测试）
@MOVF(469) D990 D502  ; 实时漏率（Pa.m3/s_Float）, #1-2腔体测试漏率（Pa.m3/s_Float）
@MOVF(469) D992 D504  ; 实时检漏口压力（Pa_Float）, #1-2腔体测试检漏口压力（Pa_Float）

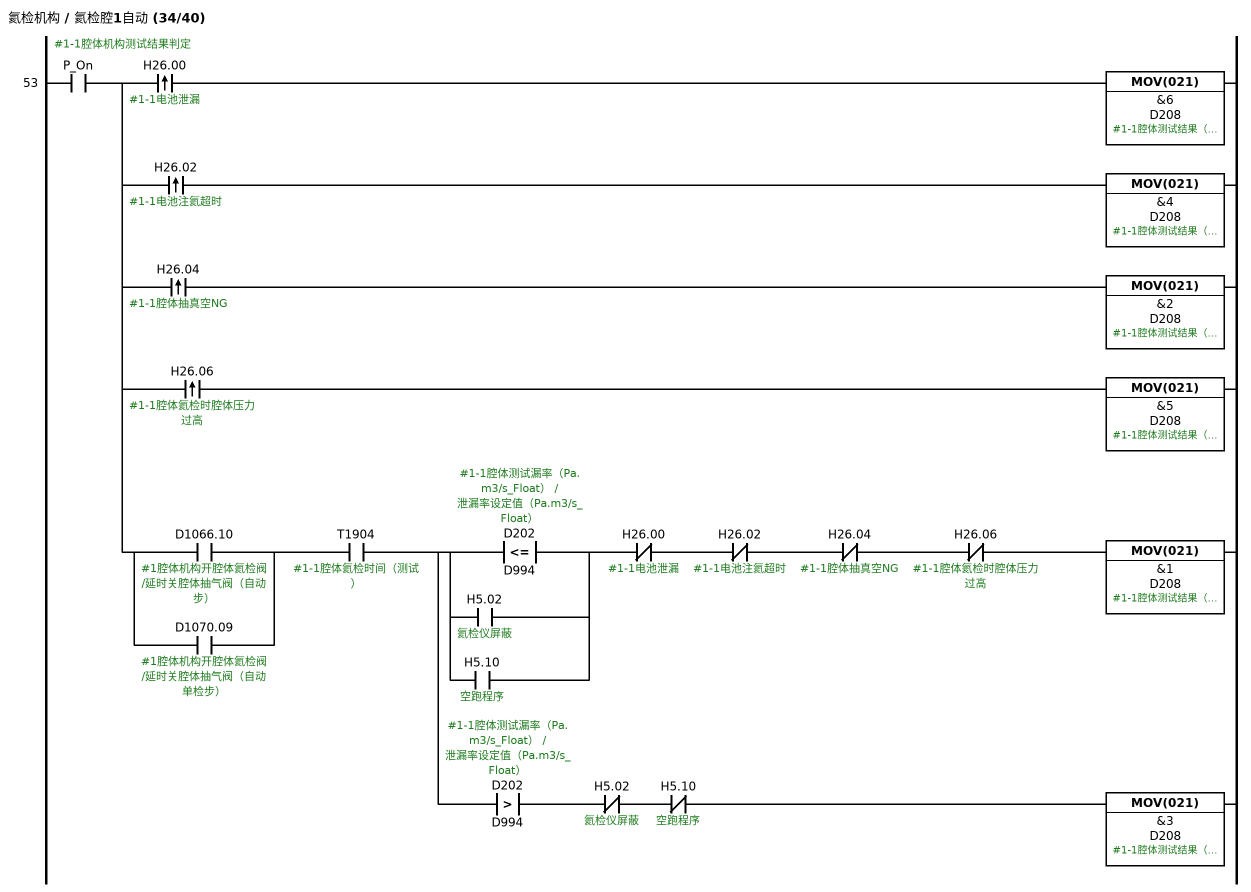
; rung 53: #1-1腔体机构测试结果判定
LD P_On
OUT TR0
@AND H26.00  ; #1-1电池泄漏
MOV(021) &6 D208  ; #1-1腔体测试结果（1 OK，2腔体泄漏，3气密NG，4注氦超时，5氦检异常，6电池泄漏）
LD TR0
@AND H26.02  ; #1-1电池注氦超时
MOV(021) &4 D208  ; #1-1腔体测试结果（1 OK，2腔体泄漏，3气密NG，4注氦超时，5氦检异常，6电池泄漏）
LD TR0
@AND H26.04  ; #1-1腔体抽真空NG
MOV(021) &2 D208  ; #1-1腔体测试结果（1 OK，2腔体泄漏，3气密NG，4注氦超时，5氦检异常，6电池泄漏）
LD TR0
@AND H26.06  ; #1-1腔体氦检时腔体压力过高
MOV(021) &5 D208  ; #1-1腔体测试结果（1 OK，2腔体泄漏，3气密NG，4注氦超时，5氦检异常，6电池泄漏）
LD TR0
LD D1066.10  ; #1腔体机构开腔体氦检阀/延时关腔体抽气阀（自动步）
OR D1070.09  ; #1腔体机构开腔体氦检阀/延时关腔体抽气阀（自动单检步）
ANDLD
AND T1904  ; #1-1腔体氦检时间（测试）
OUT TR0
LD<=F(332) D202 D994  ; #1-1腔体测试漏率（Pa.m3/s_Float）, 泄漏率设定值（Pa.m3/s_Float）
OR H5.02  ; 氦检仪屏蔽
OR H5.10  ; 空跑程序
ANDLD
ANDNOT H26.00  ; #1-1电池泄漏
ANDNOT H26.02  ; #1-1电池注氦超时
ANDNOT H26.04  ; #1-1腔体抽真空NG
ANDNOT H26.06  ; #1-1腔体氦检时腔体压力过高
MOV(021) &1 D208  ; #1-1腔体测试结果（1 OK，2腔体泄漏，3气密NG，4注氦超时，5氦检异常，6电池泄漏）
LD TR0
AND>F(333) D202 D994  ; #1-1腔体测试漏率（Pa.m3/s_Float）, 泄漏率设定值（Pa.m3/s_Float）
ANDNOT H5.02  ; 氦检仪屏蔽
ANDNOT H5.10  ; 空跑程序
MOV(021) &3 D208  ; #1-1腔体测试结果（1 OK，2腔体泄漏，3气密NG，4注氦超时，5氦检异常，6电池泄漏）

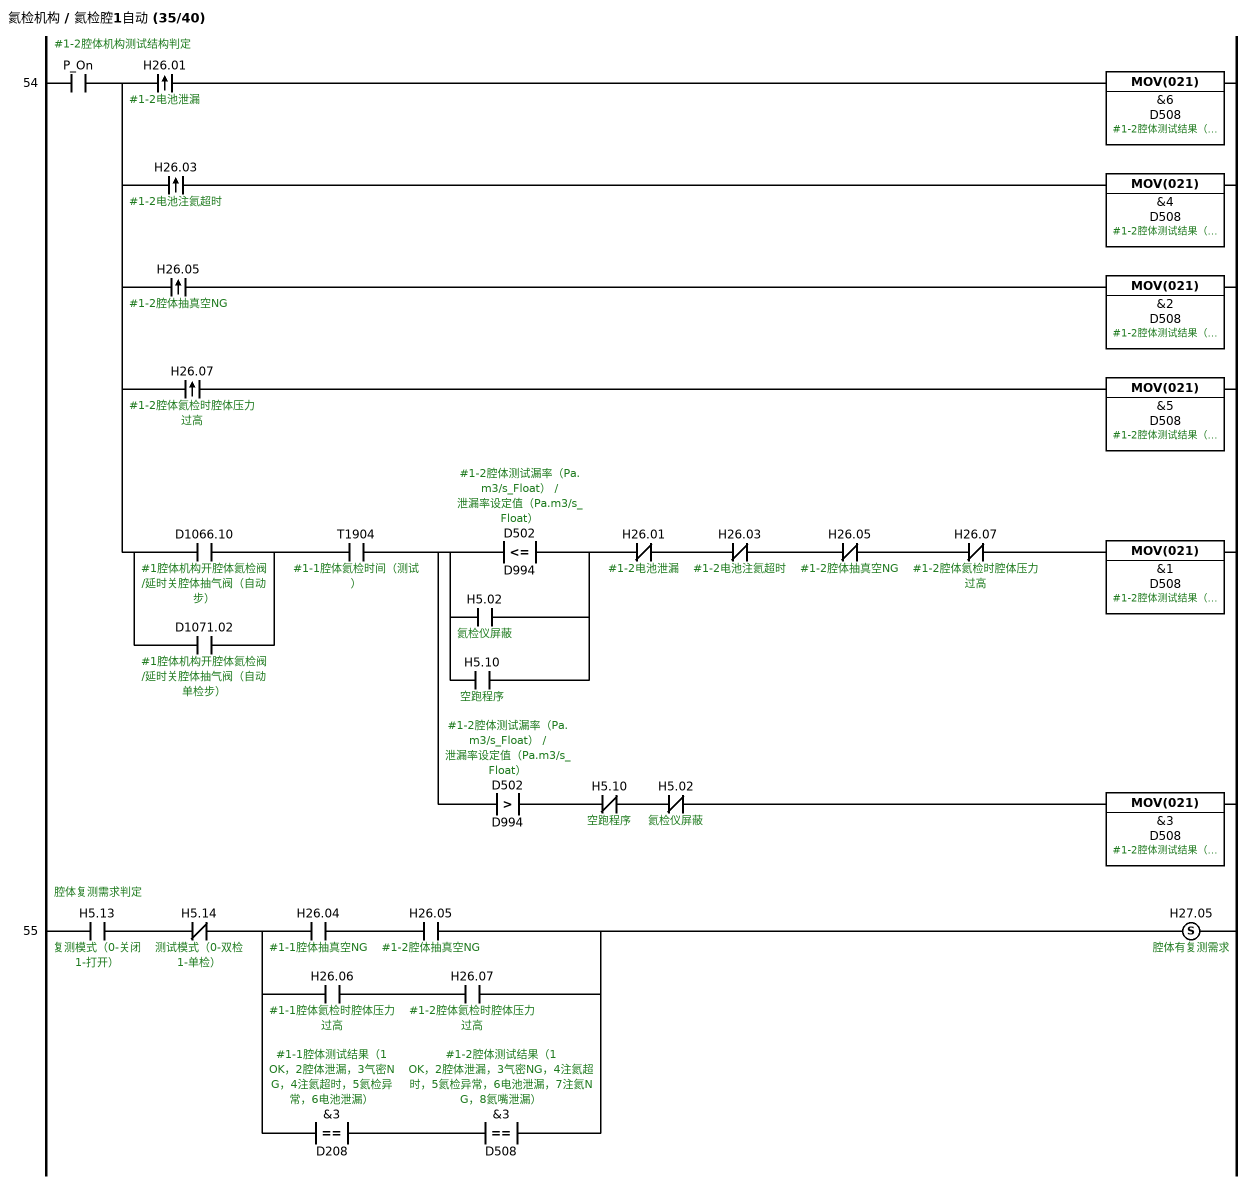
; rung 54: #1-2腔体机构测试结构判定
LD P_On
OUT TR0
@AND H26.01  ; #1-2电池泄漏
MOV(021) &6 D508  ; #1-2腔体测试结果（1 OK，2腔体泄漏，3气密NG，4注氦超时，5氦检异常，6电池泄漏，7注氦NG，8氦嘴泄漏）
LD TR0
@AND H26.03  ; #1-2电池注氦超时
MOV(021) &4 D508  ; #1-2腔体测试结果（1 OK，2腔体泄漏，3气密NG，4注氦超时，5氦检异常，6电池泄漏，7注氦NG，8氦嘴泄漏）
LD TR0
@AND H26.05  ; #1-2腔体抽真空NG
MOV(021) &2 D508  ; #1-2腔体测试结果（1 OK，2腔体泄漏，3气密NG，4注氦超时，5氦检异常，6电池泄漏，7注氦NG，8氦嘴泄漏）
LD TR0
@AND H26.07  ; #1-2腔体氦检时腔体压力过高
MOV(021) &5 D508  ; #1-2腔体测试结果（1 OK，2腔体泄漏，3气密NG，4注氦超时，5氦检异常，6电池泄漏，7注氦NG，8氦嘴泄漏）
LD TR0
LD D1066.10  ; #1腔体机构开腔体氦检阀/延时关腔体抽气阀（自动步）
OR D1071.02  ; #1腔体机构开腔体氦检阀/延时关腔体抽气阀（自动单检步）
ANDLD
AND T1904  ; #1-1腔体氦检时间（测试）
OUT TR0
LD<=F(332) D502 D994  ; #1-2腔体测试漏率（Pa.m3/s_Float）, 泄漏率设定值（Pa.m3/s_Float）
OR H5.02  ; 氦检仪屏蔽
OR H5.10  ; 空跑程序
ANDLD
ANDNOT H26.01  ; #1-2电池泄漏
ANDNOT H26.03  ; #1-2电池注氦超时
ANDNOT H26.05  ; #1-2腔体抽真空NG
ANDNOT H26.07  ; #1-2腔体氦检时腔体压力过高
MOV(021) &1 D508  ; #1-2腔体测试结果（1 OK，2腔体泄漏，3气密NG，4注氦超时，5氦检异常，6电池泄漏，7注氦NG，8氦嘴泄漏）
LD TR0
AND>F(333) D502 D994  ; #1-2腔体测试漏率（Pa.m3/s_Float）, 泄漏率设定值（Pa.m3/s_Float）
ANDNOT H5.10  ; 空跑程序
ANDNOT H5.02  ; 氦检仪屏蔽
MOV(021) &3 D508  ; #1-2腔体测试结果（1 OK，2腔体泄漏，3气密NG，4注氦超时，5氦检异常，6电池泄漏，7注氦NG，8氦嘴泄漏）
; rung 55: 腔体复测需求判定
LD H5.13  ; 复测模式（0-关闭 1-打开）
ANDNOT H5.14  ; 测试模式（0-双检 1-单检）
LD H26.04  ; #1-1腔体抽真空NG
AND H26.05  ; #1-2腔体抽真空NG
LD H26.06  ; #1-1腔体氦检时腔体压力过高
AND H26.07  ; #1-2腔体氦检时腔体压力过高
ORLD
LD=(300) &3 D208  ; #1-1腔体测试结果（1 OK，2腔体泄漏，3气密NG，4注氦超时，5氦检异常，6电池泄漏）
AND=(300) &3 D508  ; #1-2腔体测试结果（1 OK，2腔体泄漏，3气密NG，4注氦超时，5氦检异常，6电池泄漏，7注氦NG，8氦嘴泄漏）
ORLD
ANDLD
SET H27.05  ; 腔体有复测需求

